DATA_BLOCK "DB_Output"	// DB 1010
AUTHOR : Broecker
VERSION : 0.1
  STRUCT
   Spare_A100_0 : BOOL ;
   Fuse_24V_DC_Reset : BOOL ;
   Spare_A100_2 : BOOL ;
   Spare_A100_3 : BOOL ;
   Spare_A100_4 : BOOL ;
   Status_LED_Bit0 : BOOL ;
   Status_LED_Bit1 : BOOL ;
   Status_LED_Bit2 : BOOL ;
   LED_Automatic : BOOL ;
   LED_Reset : BOOL ;
   Spare_A101_2 : BOOL ;
   Spare_A101_3 : BOOL ;
   Spare_A101_4 : BOOL ;
   Spare_A101_5 : BOOL ;
   Spare_A101_6 : BOOL ;
   Spare_A101_7 : BOOL ;
   Emergency_Stop_Reset : BOOL ;
   Spare_A102_1 : BOOL ;
   Spare_A102_2 : BOOL ;
   Spare_A102_3 : BOOL ;
   Spare_A102_4 : BOOL ;
   Spare_A102_5 : BOOL ;
   Spare_A102_6 : BOOL ;
   Spare_A102_7 : BOOL ;
   Spare_A103_0 : BOOL ;
   Spare_A103_1 : BOOL ;
   Spare_A103_2 : BOOL ;
   Spare_A103_3 : BOOL ;
   Spare_A103_4 : BOOL ;
   Spare_A103_5 : BOOL ;
   Spare_A103_6 : BOOL ;
   Spare_A103_7 : BOOL ;
   Spare_A104_0 : BOOL ;
   Spare_A104_1 : BOOL ;
   Spare_A104_2 : BOOL ;
   Spare_A104_3 : BOOL ;
   Spare_A104_4 : BOOL ;
   Spare_A104_5 : BOOL ;
   Spare_A104_6 : BOOL ;
   Spare_A104_7 : BOOL ;
   Spare_A105_0 : BOOL ;
   Spare_A105_1 : BOOL ;
   Spare_A105_2 : BOOL ;
   Spare_A105_3 : BOOL ;
   Spare_A105_4 : BOOL ;
   Spare_A105_5 : BOOL ;
   Spare_A105_6 : BOOL ;
   Spare_A105_7 : BOOL ;
   Spare_A106_0 : BOOL ;
   Spare_A106_1 : BOOL ;
   Spare_A106_2 : BOOL ;
   Spare_A106_3 : BOOL ;
   Spare_A106_4 : BOOL ;
   Spare_A106_5 : BOOL ;
   Spare_A106_6 : BOOL ;
   Spare_A106_7 : BOOL ;
   Spare_A107_0 : BOOL ;
   Spare_A107_1 : BOOL ;
   Spare_A107_2 : BOOL ;
   Spare_A107_3 : BOOL ;
   Spare_A107_4 : BOOL ;
   Spare_A107_5 : BOOL ;
   Spare_A107_6 : BOOL ;
   Spare_A107_7 : BOOL ;
   Spare_A108_0 : BOOL ;
   Spare_A108_1 : BOOL ;
   Spare_A108_2 : BOOL ;
   Spare_A108_3 : BOOL ;
   Spare_A108_4 : BOOL ;
   Spare_A108_5 : BOOL ;
   Spare_A108_6 : BOOL ;
   Spare_A108_7 : BOOL ;
   Spare_A109_0 : BOOL ;
   Spare_A109_1 : BOOL ;
   Spare_A109_2 : BOOL ;
   Spare_A109_3 : BOOL ;
   Spare_A109_4 : BOOL ;
   Spare_A109_5 : BOOL ;
   Spare_A109_6 : BOOL ;
   Spare_A109_7 : BOOL ;
   Spare_A110_0 : BOOL ;
   Fuse_24V_DC_Reset_VEH : BOOL ;
   Spare_A110_2 : BOOL ;
   LED_Reset_VEH : BOOL ;
   Sound_Generator : BOOL ;
   Status_LED_Bit0_VEH : BOOL ;
   Status_LED_Bit1_VEH : BOOL ;
   Status_LED_Bit2_VEH : BOOL ;
   Emergency_Stop_Reset_VEH : BOOL ;
   Spare_A111_1 : BOOL ;
   Spare_A111_2 : BOOL ;
   Spare_A111_3 : BOOL ;
   Scanner_On : BOOL ;
   Scanner_Field_A : BOOL ;
   Scanner_Field_B : BOOL ;
   Spare_A111_7 : BOOL ;
   Spare_A112_0 : BOOL ;
   Spare_A112_1 : BOOL ;
   Safety_Bar_Op : BOOL ;
   Safety_Bar_Cl : BOOL ;
   Spare_A112_4 : BOOL ;
   Spare_A112_5 : BOOL ;
   Spare_A112_6 : BOOL ;
   Spare_A112_7 : BOOL ;
  END_STRUCT ;	
BEGIN
END_DATA_BLOCK

ORGANIZATION_BLOCK OB 1
TITLE = "Main Program Sweep (Cycle)"
VERSION : 0.1
VAR_TEMP
  OB1_EV_CLASS : BYTE ;	//Bits 0-3 = 1 (Coming event), Bits 4-7 = 1 (Event class 1)
  OB1_SCAN_1 : BYTE ;	//1 (Cold restart scan 1 of OB 1), 3 (Scan 2-n of OB 1)
  OB1_PRIORITY : BYTE ;	//Priority of OB Execution
  OB1_OB_NUMBR : BYTE ;	//1 (Organization block 1, OB1)
  OB1_RESERVED_1 : BYTE ;	//Reserved for system
  OB1_RESERVED_2 : BYTE ;	//Reserved for system
  OB1_PREV_CYCLE : INT ;	//Cycle time of previous OB1 scan (milliseconds)
  OB1_MIN_CYCLE : INT ;	//Minimum cycle time of OB1 (milliseconds)
  OB1_MAX_CYCLE : INT ;	//Maximum cycle time of OB1 (milliseconds)
  OB1_DATE_TIME : DATE_AND_TIME ;	//Date and time OB1 started
END_VAR
BEGIN
// (block stored without names or comments; labels and parameter names are numbered)
END_ORGANIZATION_BLOCK

SYMBOL_TABLE
"IDB_Safe_Main"	DB 1	FB 1
"DB_TRO"	DB 2	DB 2
"DB_LIF"	DB 3	DB 3
"DB_TEL"	DB 4	DB 4
"DB_BRI"	DB 5	DB 5
"DB_ComGateway"	DB 10	DB 10
"IDB_FB2_TRO"	DB 12	FB 2
"IDB_FB2_LIF"	DB 13	FB 2
"IDB_FB21_TEL"	DB 14	FB 21
"DB_OrderBuffer"	DB 15	DB 15
"DB_IntentData"	DB 17	DB 17
"DB_TargetData"	DB 19	DB 19
"IDB_FB22"	DB 22	FB 22
"IDB_FB29"	DB 29	FB 29
"IDB_MasterInterface"	DB 33	FB 13
"DB_ANALOG"	DB 50	DB 50
"INOUT"	DB 80	DB 80
"DB_ActualHookdata"	DB 92	DB 92	// Hookdata of actual trollayposition
"Moves"	DB 101	DB 101
"InstanzDB PNIODiag"	DB 126	FB 126
"InstanzDB STATDiag"	DB 127	DB 127
"DB_Crane"	DB 130	DB 130
"DB_Steps"	DB 132	DB 132
"DB_CylinderTypes"	DB 133	DB 133
"IDB_FB190"	DB 190	FB 190
"IDB_FB190_2"	DB 191	FB 190
"IDB1_FB192"	DB 192	FB 192
"IDB1_FB192_2"	DB 193	FB 192
"TRO_Positions"	DB 200	DB 200
"BR01_TR01"	DB 201	DB 201
"BR01_TR02"	DB 202	DB 202
"BR01_TR03"	DB 203	DB 203
"BR01_TR04"	DB 204	DB 204
"BR01_TR05"	DB 205	DB 205
"BR01_TR06"	DB 206	DB 206
"BR01_TR07"	DB 207	DB 207
"BR01_TR08"	DB 208	DB 208
"BR01_TR09"	DB 209	DB 209
"BR01_TR10"	DB 210	DB 210
"BR01_TR11"	DB 211	DB 211
"BR02_TR01"	DB 212	DB 212
"BR02_TR02"	DB 213	DB 213
"BR02_TR03"	DB 214	DB 214
"BR02_TR04"	DB 215	DB 215
"BR02_TR05"	DB 216	DB 216
"BR02_TR06"	DB 217	DB 217
"BR02_TR07"	DB 218	DB 218
"BR02_TR08"	DB 219	DB 219
"BR02_TR09"	DB 220	DB 220
"BR02_TR10"	DB 221	DB 221
"BR02_TR11"	DB 222	DB 222
"BR03_TR01"	DB 223	DB 223
"BR03_TR02"	DB 224	DB 224
"BR03_TR03"	DB 225	DB 225
"BR03_TR04"	DB 226	DB 226
"BR03_TR05"	DB 227	DB 227
"BR03_TR06"	DB 228	DB 228
"BR03_TR07"	DB 229	DB 229
"BR03_TR08"	DB 230	DB 230
"BR03_TR09"	DB 231	DB 231
"BR03_TR10"	DB 232	DB 232
"BR03_TR11"	DB 233	DB 233
"BR04_TR01"	DB 234	DB 234
"BR04_TR02"	DB 235	DB 235
"BR04_TR03"	DB 236	DB 236
"BR04_TR04"	DB 237	DB 237
"BR04_TR05"	DB 238	DB 238
"BR04_TR06"	DB 239	DB 239
"BR04_TR07"	DB 240	DB 240
"BR04_TR08"	DB 241	DB 241
"BR04_TR09"	DB 242	DB 242
"BR04_TR10"	DB 243	DB 243
"BR04_TR11"	DB 244	DB 244
"BR05_TR01"	DB 245	DB 245
"BR05_TR02"	DB 246	DB 246
"BR05_TR03"	DB 247	DB 247
"BR05_TR04"	DB 248	DB 248
"BR05_TR05"	DB 249	DB 249
"BR05_TR06"	DB 250	DB 250
"BR05_TR07"	DB 251	DB 251
"BR05_TR08"	DB 252	DB 252
"BR05_TR09"	DB 253	DB 253
"BR05_TR10"	DB 254	DB 254
"BR05_TR11"	DB 255	DB 255
"BR06_TR01"	DB 256	DB 256
"BR06_TR02"	DB 257	DB 257
"BR06_TR03"	DB 258	DB 258
"BR06_TR04"	DB 259	DB 259
"BR06_TR05"	DB 260	DB 260
"BR06_TR06"	DB 261	DB 261
"BR06_TR07"	DB 262	DB 262
"BR06_TR08"	DB 263	DB 263
"BR06_TR09"	DB 264	DB 264
"BR06_TR10"	DB 265	DB 265
"BR06_TR11"	DB 266	DB 266
"BR07_TR01"	DB 267	DB 267
"BR07_TR02"	DB 268	DB 268
"BR07_TR03"	DB 269	DB 269
"BR07_TR04"	DB 270	DB 270
"BR07_TR05"	DB 271	DB 271
"BR07_TR06"	DB 272	DB 272
"BR07_TR07"	DB 273	DB 273
"BR07_TR08"	DB 274	DB 274
"BR07_TR09"	DB 275	DB 275
"BR07_TR10"	DB 276	DB 276
"BR07_TR11"	DB 277	DB 277
"BR08_TR01"	DB 278	DB 278
"BR08_TR02"	DB 279	DB 279
"BR08_TR03"	DB 280	DB 280
"BR08_TR04"	DB 281	DB 281
"BR08_TR05"	DB 282	DB 282
"BR08_TR06"	DB 283	DB 283
"BR08_TR07"	DB 284	DB 284
"BR08_TR08"	DB 285	DB 285
"BR08_TR09"	DB 286	DB 286
"BR08_TR10"	DB 287	DB 287
"BR08_TR11"	DB 288	DB 288
"BR09_TR01"	DB 289	DB 289
"BR09_TR02"	DB 290	DB 290
"BR09_TR03"	DB 291	DB 291
"BR09_TR04"	DB 292	DB 292
"BR09_TR05"	DB 293	DB 293
"BR09_TR06"	DB 294	DB 294
"BR09_TR07"	DB 295	DB 295
"BR09_TR08"	DB 296	DB 296
"BR09_TR09"	DB 297	DB 297
"BR09_TR10"	DB 298	DB 298
"BR09_TR11"	DB 299	DB 299
"BR10_TR01"	DB 300	DB 300
"BR10_TR02"	DB 301	DB 301
"BR10_TR03"	DB 302	DB 302
"BR10_TR04"	DB 303	DB 303
"BR10_TR05"	DB 304	DB 304
"BR10_TR06"	DB 305	DB 305
"BR10_TR07"	DB 306	DB 306
"BR10_TR08"	DB 307	DB 307
"BR10_TR09"	DB 308	DB 308
"BR10_TR10"	DB 309	DB 309
"BR10_TR11"	DB 310	DB 310
"BR11_TR01"	DB 311	DB 311
"BR11_TR02"	DB 312	DB 312
"LIF_Pos"	DB 350	DB 350
"IDB_Modbus1"	DB 362	FB 102
"ProfiNet"	DB 400	DB 400
"Error_Safety"	DB 410	DB 410
"IDB_ESTOP_1"	DB 450	FB 215
"IDB_ESTOP_2"	DB 451	FB 185
"IDB_Auto"	DB 452	FB 186
"F_GLOBDB"	DB 545	DB 545	// F_: F_Global_Data Block
"F00035_75x_667_4FDI_4FDO"	DB 555	FB 272
"F00040_75x_667_4FDI_4FDO"	DB 556	FB 272
"F00045_75x_661_4FDI_24V"	DB 557	FB 272
"F00055_75x_667_4FDI_4FDO"	DB 558	FB 272
"F_IO"	DB 690	DB 690
"F_Position"	DB 695	DB 695
"F_GBL_RECV"	DB 750	DB 750
"IDB_F_RCV"	DB 751	FB 226
"F_GBL_SEND"	DB 752	DB 752
"IDB_F_SND"	DB 753	FB 225
"IDB_WagoiPar_Rack"	DB 901	FB 37
"IDB_WagoiPar_BRI"	DB 920	FB 37
"IDB_WagoiPar_TRO"	DB 921	FB 37
"IDB_WagoiPar_LIF"	DB 922	FB 37
"DB_iPar_Diag"	DB 930	FB 101
"DIAG_PROFI_V2_iPar"	DB 931	DB 931	// diagnosis data of PROFIsafe modules V2 iPar with FB101
"DB_Vorlage"	DB 999	DB 999
"DB_LS1"	DB 1300	DB 1300
"IDB_LS1_Circum"	DB 1329	FB 29
"DB_LS"	DB 1350	DB 1350
"iPar_Data_Rack"	DB 1901	DB 1901
"iPar_Data_Bridge"	DB 1920	DB 1920
"iPar_Data_Trolley"	DB 1921	DB 1921
"iPar_Data_Lift"	DB 1922	DB 1922
"Safe_Main"	FB 1	FB 1
"MovidriveB_Control"	FB 2	FB 2
"MasterInterface"	FB 13	FB 13
"CheckEncoder"	FB 21	FB 21
"GetCircumference"	FB 22	FB 22
"WAGO_Analog_Input_4_20"	FB 29	FB 29	// WAGO A/D-Wandler 4-20mA
"WAGO_iPar_UDL_4_Mod"	FB 37	FB 37	// WAGO up- / download iParameter PROFIsafe Modules
"TSEND"	FB 63	FB 63	// Send Data
"TRCV"	FB 64	FB 64	// Receive Data
"TCON"	FB 65	FB 65	// Connect
"TDISCON"	FB 66	FB 66	// Disconnect
"Safety_Position"	FB 70	FB 70	// Sichere Positionsüberwachung
"Safety_Direction"	FB 72	FB 72	// Sichere Richtungserfassung
"Safety_Speed"	FB 73	FB 73	// Sichere Geschwindigkeit
"Safety_SpeedCheck"	FB 74	FB 74
"Wago_Trolley"	FB 81	FB 81
"F_Input_MAP"	FB 91	FB 91
"ESTOP"	FB 92	FB 92
"GetArea"	FB 95	FB 95
"DiagPROFIsafe_V2_iPar"	FB 101	FB 101	// read diagnosis data of PROFIsafe modules V2 iPar
"MODBUSPN"	FB 102	FB 102	// MODBUS PN CPU
"TCP_COMM"	FB 103	FB 103	// TCP Kommunikation
"MOD_CLI"	FB 104	FB 104
"MOD_SERV"	FB 105	FB 105
"PNIODiag"	FB 126	FB 126	// Profibus/DP und Profinet/IO-Diagnose
"STATDiag"	FB 127	FB 127	// Zweitbaustein (PNIODiag)
"F_TON"	FB 185	FB 185	// F_: Timer Switch On Delay
"F_TOF"	FB 186	FB 186	// F_: Timer Switch Off Delay
"CopyHookDBs"	FB 190	FB 190
"READ_DBL"	FB 192	FB 192	// read db from memorycard
"WRITE_DBL"	FB 193	FB 193	// write db to memorycard
"F_ESTOP1"	FB 215	FB 215	// F_: Emergency Stop / Stop Category 1
"F_ACK_GL"	FB 219	FB 219	// F_: Global Acknowledgement of all F-I/O of a RTG
"F_SENDS7"	FB 225	FB 225	// F_: Send S7 Connection
"F_RCVS7"	FB 226	FB 226	// F_: Receive S7 Connection
"F_IO_CGP"	FB 272	FB 272	// F_: Driver Block In-Output with Channel Granular Passivation
"F_CTRL_1"	FB 273	FB 273
"F_CTRL_2"	FB 274	FB 274	// F_: Test Block an Programm Run Control
"F_DIAG_N"	FB 275	FB 275
"FITON"	FB 276	FB 276
"FITOF"	FB 277	FB 277
"FIACK_GL"	FB 278	FB 278
"F-CALL"	FC 1	FC 1
"Init"	FC 2	FC 2
"AG_SEND"	FC 5	FC 5	// AG SEND
"AG_RECV"	FC 6	FC 6	// AG RECEIVE
"DT_TOD"	FC 8	FC 8	// DT to TOD
"OpHours"	FC 9	FC 9
"EQ_STRNG"	FC 10	FC 10	// Equal String
"AbsEncoder"	FC 11	FC 11
"Motor_2_frequ"	FC 12	FC 12
"DT to DATE"	FC 15	FC 15	// DT to DATE
"Scan_BRI"	FC 21	FC 21
"Scan_BRI_MAN"	FC 22	FC 22	// Scan Bride Manual Mode
"Scan_BRI_DBs"	FC 23	FC 23
"Scan_LIF"	FC 25	FC 25
"Scan_LIF_Man"	FC 26	FC 26
"Scan_TEL"	FC 27	FC 27
"Scan_TEL_Man"	FC 28	FC 28
"SCALE_WAGO_AI"	FC 29	FC 29	// for WAGO 250-466 4-20mA SE Standard
"Inputs"	FC 30	FC 30
"Outputs"	FC 31	FC 31
"MeasureSystem"	FC 33	FC 33
"SEL"	FC 36	FC 36	// Select
"Errors"	FC 40	FC 40
"Errors Reset"	FC 41	FC 41
"Errors_001-016_GEN1"	FC 42	FC 42
"Errors_017-032_GEN2"	FC 43	FC 43
"Errors_033-048_NET"	FC 44	FC 44
"Errors_113-128"	FC 45	FC 45
"Errors_129-144_08"	FC 46	FC 46
"Errors_145-160"	FC 47	FC 47
"EOff_MachineOff"	FC 48	FC 48
"OP_Mode"	FC 49	FC 49
"Send_Buffer"	FC 52	FC 52
"MSG_161-176"	FC 55	FC 55
"MSG_177_192"	FC 56	FC 56
"CableDrum"	FC 60	FC 60
"TargetPosLift"	FC 70	FC 70
"CheckHookType"	FC 72	FC 72
"CheckWindowDi"	FC 100	FC 100
"Communication"	FC 103	FC 103
"STEPS_Control"	FC 110	FC 110
"STEPS_OrderData"	FC 111	FC 111
"STEPS_BASEPOS"	FC 112	FC 112
"STEPS_EMPTY"	FC 113	FC 113
"STEPS_GET"	FC 114	FC 114
"STEPS_PUT"	FC 115	FC 115
"Axis_TROLLEY"	FC 210	FC 210
"Axis_TROLLEY_Release"	FC 211	FC 211
"Axis_TROLLEY_Control"	FC 212	FC 212
"Axis_TROLLEY_Speed"	FC 213	FC 213
"Axis_TROLLEY_Scan"	FC 214	FC 214
"Axis_TROLLEY_Scan_Man"	FC 215	FC 215
"Axis_TROLLEY_Flt_065-080"	FC 219	FC 219
"Axis_LIFT"	FC 220	FC 220
"Axis_LIFT_Control"	FC 222	FC 222
"Axis_LIFT_Speed"	FC 223	FC 223
"Axis_LIFT_Scan"	FC 224	FC 224
"Axis_LIFT_Flt_081-096"	FC 229	FC 229
"Axis_TELESCOPES"	FC 230	FC 230
"Axis_TEL_Control"	FC 232	FC 232
"Axis_TEL_Speed"	FC 233	FC 233
"Axis_TEL_Scan"	FC 234	FC 234
"Axis_TEL_Chk"	FC 235	FC 235
"Axis_TEL_Status"	FC 236	FC 236
"Axis_TEL_Mode_Status"	FC 237	FC 237
"Axis_TEL_BCD"	FC 238	FC 238
"Axis_TEL_Flt_097-112"	FC 239	FC 239
"Axis_TEL_Encoder"	FC 240	FC 240
"iPar_ServerCall"	FC 900	FC 900
"Scan_LIF_New"	FC 1025	FC 1025
"Scan_LIF_Man_New"	FC 1026	FC 1026
"TROGetPosVal"	FC 1071	FC 1071
"E   35.0"	I 35.0	BOOL	// spare
"E   35.1"	I 35.1	BOOL	// spare
"I_TRO_FB_Lift"	I 35.2	BOOL	// Feedback safestop lift
"I_TRO_FB_Trolley"	I 35.3	BOOL	// Feedback safestop  trolley
"I_TRO_FB_Telescope"	I 40.0	BOOL	// Feedback safestop no FU
"E   40.1"	I 40.1	BOOL	// spare
"I_TRO_FB_Estop_CH1"	I 40.2	BOOL	// Feedback E-Stop  CH1
"I_TRO_FB_Estop_CH2"	I 40.3	BOOL	// Feedback E-Stop  CH2
"I_TRO_EStop"	I 45.0	BOOL	// Emergency stop activ
"I_TRO_Brake_OK"	I 45.1	BOOL	// Temperature brake resistors OK
"E   45.2"	I 45.2	BOOL	// spare
"E   45.3"	I 45.3	BOOL	// spare
"I_TRO_LIF_Overl_L_NC"	I 55.0	BOOL	// Overload-Monitoring left NC
"I_TRO_LIF_Overl_R_NC"	I 55.1	BOOL	// Overload-Monitoring right NC
"I_TRO_LIF_Slap_L_NC"	I 55.2	BOOL	// Slap-Rope-Monitoring left NC
"I_TRO_LIF_Slap_R_NC"	I 55.3	BOOL	// Slap-Rope-Monitoring right NC
"I_TRO_Fuse_115V_OK"	I 75.0	BOOL	// 115V AC OK
"I_TRO_Fuse_24V_OK"	I 75.1	BOOL	// fuse 24V DC OK
"I_TRO_Overtemp_Cabinet"	I 75.2	BOOL	// high temperature cabinet
"I_TRO_Power Brakes_OK"	I 75.3	BOOL	// Power supply brakes OK
"I_TRO_Power_Lift_OK"	I 75.4	BOOL	// Power supply lift OK
"I_TRO_Power_Drum_OK"	I 75.5	BOOL	// Power supply cable drum OK
"I_TRO_Power_Cabinet_Fan"	I 75.6	BOOL	// Power supply cabinet fan OK
"I_TRO_Cabinet_Fan_On"	I 75.7	BOOL	// cabinet fan running
"I_TRO_BTN_Reset"	I 76.0	BOOL	// Reset button (top cabinet)
"I_TRO_BTN_Preset"	I 76.1	BOOL	// Preset button (3s)
"I_TRO_Preset_Bit_0"	I 76.2	BOOL	// Preset selection switch bit 0
"I_TRO_Preset_Bit_1"	I 76.3	BOOL	// Preset selection switch bit 1
"I_TRO_Preset_Bit_2"	I 76.4	BOOL	// Preset selection switch bit 2
"I_TRO_Preset_Bit_3"	I 76.5	BOOL	// Preset selection switch bit 3
"E 76_6"	I 76.6	BOOL	// spare
"E 76_7"	I 76.7	BOOL	// spare
"I_Check_CableDrum_NO"	I 77.0	BOOL	// check cable drum NO
"I_Check_CableDrum_NC"	I 77.1	BOOL	// check cable drum NC
"E  77_2"	I 77.2	BOOL	// spar
"E  77_3"	I 77.3	BOOL	// spar
"I_Buffer_left_Free"	I 77.4	BOOL	// Buffer left occupied //
"I_Buffer_right_Free"	I 77.5	BOOL	// Buffer right occupied //
"I_LIF_Limit_TOP"	I 77.6	BOOL	// Lift limit switch top (minus)
"I_LIF_Limit_BOTTOM"	I 77.7	BOOL	// Lift limit switch bottom (plus)
"I_LIF_Pos_TOP_NO"	I 78.0	BOOL	// Lift limit prox. top NO
"I_LIF_Pos_TOP_NC"	I 78.1	BOOL	// Lift limit prox. top NC
"I_TRO_Limit_plus"	I 78.2	BOOL	// Tolley limit switch plus
"I_TRO_Limit_minus"	I 78.3	BOOL	// Tolley limit switch minus
"I_TRO_FS_plus_NO"	I 78.4	BOOL	// Tolley prox. switch forced slow plus NO
"I_TRO_FS_plus_NC"	I 78.5	BOOL	// Tolley prox. switch forced slow plus NC
"I_TRO_FS_minus_NO"	I 78.6	BOOL	// Tolley prox. switch forced slow minus NO
"I_TRO_FS_minus_NC"	I 78.7	BOOL	// Tolley prox. switch forced slow minus NC
"I_SSI_Barcode_noPos"	I 79.0	BOOL	// Datamatrix SSI error: no position
"I_SSI_Barcode_dirty"	I 79.1	BOOL	// Datamatrix SSI error: dirty
"I_Profinet_Barcode_noPos"	I 79.2	BOOL	// Datamatrix Profinet error: no position
"I_Profinet_Barcode_dirty"	I 79.3	BOOL	// Datamatrix Profinet error: dirty
"I_TRO_Drop_1_P"	I 79.4	BOOL	// Trolley drop off protection plus 1
"I_TRO_Drop_2_P"	I 79.5	BOOL	// Trolley drop off protection plus 2
"I_TRO_Drop_1_M"	I 79.6	BOOL	// Trolley drop off protection minus 1
"I_TRO_Drop_2_M"	I 79.7	BOOL	// Trolley drop off protection minus 2
"I_TRO_Plus"	I 80.0	BOOL	// Trolley drive plus
"I_TRO_Minus"	I 80.1	BOOL	// Trolley drive minus
"I_Lift_up"	I 80.2	BOOL	// Lift drive up
"I_Lift_down"	I 80.3	BOOL	// Lift drive down
"I_TEL_Plus"	I 80.4	BOOL	// Tellescope drive plus
"I_TEL_Minus"	I 80.5	BOOL	// Telescope drive minus
"E 80_6"	I 80.6	BOOL	// spare
"E 80_7"	I 80.7	BOOL	// spare
"E 85_0"	I 85.0	BOOL	// spare
"E 85_1"	I 85.1	BOOL	// spare
"E 85_2"	I 85.2	BOOL	// spare
"E 85_3"	I 85.3	BOOL	// spare
"I_TEL_Status1"	I 85.4	BOOL	// Drive telescopes status1
"I_TEL_Status2"	I 85.5	BOOL	// Drive telescopes status2
"E 85_6"	I 85.6	BOOL
"E 85_7"	I 85.7	BOOL
"I_LIF_Overload_L_NO"	I 86.0	BOOL	// Overload-Monitoring left NO
"I_LIF_Overload_R_NO"	I 86.1	BOOL	// Overload-Monitoring right NO
"I_LIF_SlapRope_L_NO"	I 86.2	BOOL	// Slap-Rope-Monitoring left NO
"I_LIF_SlapRope_R_NO"	I 86.3	BOOL	// Slap-Rope-Monitoring right NO
"E      86.4"	I 86.4	BOOL	// spare
"E      86.5"	I 86.5	BOOL	// spare
"I_LIF_Front_LastHookOcc"	I 86.6	BOOL	// hook front left occupied long
"I_LIF_Front_FirstHookOcc"	I 86.7	BOOL	// hook rear left occupied short
"I_LIF_Rear_LastHookOcc"	I 87.0	BOOL	// hook front right occupied long
"I_LIF_Rear_FirstHookOcc"	I 87.1	BOOL	// hook rear right occupied short
"E      87.2"	I 87.2	BOOL	// spare
"E      87.3"	I 87.3	BOOL	// spare
"I_TEL_inMidle_L"	I 87.4	BOOL	// telescope left in middle position
"I_TEL_inMidle_R"	I 87.5	BOOL	// telescope right in middle position
"E      87.6"	I 87.6	BOOL
"I_TEL_Left_Occ_NO"	I 87.7	BOOL	// telescope left occupied NO
"E      88.0"	I 88.0	BOOL
"I_TEL_Right_Occ_NO"	I 88.1	BOOL	// telescope right occupied NO
"I_TEL_Limit_front_NO"	I 88.2	BOOL	// telescopes limit switch front NO
"I_TEL_Limit_front_NC"	I 88.3	BOOL	// telescopes limit switch front NC
"I_TEL_Limit_back_NO"	I 88.4	BOOL	// telescopes limit switch back NO
"I_TEL_Limit_back_NC"	I 88.5	BOOL	// telescopes limit switch back NC
"E      88.6"	I 88.6	BOOL	// spare
"E      88.7"	I 88.7	BOOL	// spare
"E      89.0"	I 89.0	BOOL
"E      89.1"	I 89.1	BOOL
"E      89.2"	I 89.2	BOOL
"E      89.3"	I 89.3	BOOL
"E      89.4"	I 89.4	BOOL
"E      89.5"	I 89.5	BOOL
"E      89.6"	I 89.6	BOOL
"E      89.7"	I 89.7	BOOL
"OFF"	M 0.0	BOOL	// immer aus
"ON"	M 0.1	BOOL	// immer ein
"TRUE"	M 0.2	BOOL
"FALSE"	M 0.3	BOOL
"FIRST_RUN"	M 0.7	BOOL
"ModeService"	M 1.0	BOOL
"ModeManual"	M 1.1	BOOL
"ModeAuto"	M 1.2	BOOL
"ModeBypass"	M 1.3	BOOL
"ModeServiceOrManual"	M 1.4	BOOL
"SEW_EmergencyMode"	M 1.5	BOOL
"ModeAutoOrManual"	M 1.6	BOOL
"LifeBitMasterOK"	M 1.7	BOOL
"Eoff"	M 2.0	BOOL
"DivEoff"	M 2.1	BOOL
"Error"	M 2.2	BOOL
"EmOffRelais_delayed"	M 3.0	BOOL
"TRO_pFL_StopOnCarrier"	M 8.0	BOOL
"TRO_StopOnCarrier"	M 8.1	BOOL
"LIF_pFl_manPrevPos"	M 9.0	BOOL
"LIF_pFl_manNextPos"	M 9.1	BOOL
"Tel_pFl_manMinusPos"	M 9.2	BOOL
"Tel_pFl_manPlusPos"	M 9.3	BOOL
"TEL_nFl_CenterPos"	M 9.4	BOOL
"TEL_StopInCenter"	M 9.5	BOOL
"TEL_pFl_StopInCenter"	M 9.6	BOOL
"Clock0_1"	M 10.0	BOOL	// CPU-Takt 0,1s
"Clock0_2"	M 10.1	BOOL	// CPU-Takt 0,2s
"Clock0_4"	M 10.2	BOOL	// CPU-Takt 0,4s
"Clock0_5"	M 10.3	BOOL	// CPU-Takt 0,5s
"Clock0_8"	M 10.4	BOOL	// CPU-Takt 0,8s
"Clock1_0"	M 10.5	BOOL	// CPU-Takt 1,0s
"Clock1_6"	M 10.6	BOOL	// CPU-Takt 1,6s
"Clock2_0"	M 10.7	BOOL	// CPU-Takt 2,0s
"Tick0_1"	M 11.0	BOOL	// Impuls 0,1s
"Tick0_2"	M 11.1	BOOL	// Impuls 0,2s
"Tick0_4"	M 11.2	BOOL	// Impuls 0,4s
"Tick0_5"	M 11.3	BOOL	// Impuls 0,6s
"Tick0_8"	M 11.4	BOOL	// Impuls 0,8s
"Tick1_0"	M 11.5	BOOL	// Impuls 1,0s
"Tick1_6"	M 11.6	BOOL	// Impuls 1,6s
"Tick2_0"	M 11.7	BOOL	// Impuls 2,0s
"SysPulse_0_1"	M 12.0	BOOL
"SysPulse_0_2"	M 12.1	BOOL
"SysPulse_0_4"	M 12.2	BOOL
"SysPulse_0_5"	M 12.3	BOOL
"SysPulse_0_8"	M 12.4	BOOL
"SysPulse_1_0"	M 12.5	BOOL
"SysPulse_1_6"	M 12.6	BOOL
"SysPulse_2_0"	M 12.7	BOOL
"StartModeAuto"	M 13.0	BOOL
"TEL_pFl_Start"	M 19.0	BOOL
"NullBit"	M 20.0	BOOL
"CB_Lamp_Preset"	M 21.0	BOOL
"TEL_Save_Long_POS_front"	M 25.0	BOOL
"TEL_Save_Long_POS_rear"	M 25.1	BOOL
"TrolleyWasOnCarrier"	M 40.0	BOOL
"SendTrolleyWasOnCarrier"	M 40.1	BOOL
"Next_Step"	M 44.0	BOOL
"SingleStep_ON"	M 44.1	BOOL
"One_Single_Step"	M 44.2	BOOL
"TEL_RackPos"	M 55.0	BOOL
"TEL_LS1_Pos"	M 55.1	BOOL
"TEL_LS2_Pos"	M 55.2	BOOL
"TEL_LS3_Pos"	M 55.3	BOOL
"Safety_Tele_Center"	M 152.0	BOOL
"Safety_Tele_Rear"	M 152.1	BOOL
"Safety_Tele_Front"	M 152.2	BOOL
"Safety_Trolley_in_Pos"	M 153.0	BOOL
"Safety_Lift_Top"	M 154.0	BOOL
"Safety_Lift_Over"	M 154.1	BOOL
"Safety_Lift_Under"	M 154.2	BOOL
"Mode_Bypass"	M 200.2	BOOL
"RED_IBN_Test"	M 420.0	BOOL
"IBN_1"	M 500.0	BOOL
"IBN_0"	M 500.1	BOOL
"TRO_iPar_Check"	M 921.0	BOOL
"TRO_iPar_UpLoad"	M 921.1	BOOL
"TRO_iPar_DownL"	M 921.2	BOOL
"TRO_iPar_ReqDiag"	M 921.5	BOOL
"LIF_iPar_Check"	M 922.0	BOOL
"LIF_iPar_UpLoad"	M 922.1	BOOL
"LIF_iPar_DownL"	M 922.2	BOOL
"LIF_iPar_ReqDiag"	M 922.5	BOOL
"TRO_pFl_iPar"	M 925.1	BOOL
"LIF_pFl_iPar_1"	M 925.2	BOOL
"LIF_pFl_iPar_2"	M 925.3	BOOL
"PowerFan_pl"	M 1001.0	BOOL
"PowerFan_n"	M 1001.1	BOOL
"P_FL_TeleCheck1"	M 1401.2	BOOL
"N_FL_TeleCheck1"	M 1401.3	BOOL
"P_FL_TeleCheck2"	M 1401.6	BOOL
"N_FL_TeleCheck2"	M 1401.7	BOOL
"TeleCheckErr1"	M 1402.0	BOOL
"TeleCheckErr2"	M 1402.1	BOOL
"TeleCheckErr3"	M 1402.3	BOOL
"TeleCheckErr4"	M 1402.4	BOOL
"Reset_Err"	M 1410.0	BOOL
"Impuls_1"	M 1500.0	BOOL
"Impuls_2"	M 1500.1	BOOL
"Impuls_3"	M 1500.2	BOOL
"Impuls_4"	M 1500.3	BOOL
"Impuls_5"	M 1500.4	BOOL
"Impuls_6"	M 1500.5	BOOL
"Impuls_7"	M 1500.6	BOOL
"Impuls_8"	M 1500.7	BOOL
"Bruno_B1"	M 2013.0	BOOL	// Programmpunkt muss noch bearbeitet werden
"Bruno_B2"	M 2013.1	BOOL	// Schmiermerker
"TEL_SaveTarget"	MW 14	INT
"NullWord"	MW 20	WORD
"PC_MSG_Counter"	MW 120	INT
"Bruno_W1"	MW 2014	WORD	// Schmierwort
"Bruno_W2"	MW 2016	WORD	// Schmierwort
"CYCL_EXC"	OB 1	OB 1
"CYC_INT5"	OB 35	OB 35	// Cyclic Interrupt 5
"CYCL_FLT"	OB 80	OB 80	// Cycle Time Fault
"I/O_FLT1"	OB 82	OB 82	// I/O Point Fault 1
"I/O_FLT2"	OB 83	OB 83	// I/O Point Fault 2
"OBNL_FLT"	OB 85	OB 85	// OB Not Loaded Fault
"RACK_FLT"	OB 86	OB 86	// Loss of Rack Fault
"COMM_FLT"	OB 87	OB 87	// Communication Fault
"STARTUP"	OB 100	OB 100
"PROG_ERR"	OB 121	OB 121	// Programming Error
"MOD_ERR"	OB 122	OB 122	// Module Access Error
"O_Bypass_RC"	Q 35.0	BOOL	// bypass remote control
"A    35.1"	Q 35.1	BOOL	// spare
"O_SafeStop_Lift"	Q 35.2	BOOL	// safe stop lift
"O_SafeStop_Trolley"	Q 35.3	BOOL	// safe stop trolley
"O_SafeStop_Telecope"	Q 40.0	BOOL	// safe stop telescope
"A    40.1"	Q 40.1	BOOL	// spare
"O_TRO_Stop_CH1"	Q 40.2	BOOL	// E-Stop trolley CH1
"O_TRO_Stop_CH2"	Q 40.3	BOOL	// E-Stop trolley CH2
"O_SafeRelease_Telescope"	Q 55.0	BOOL
"A 75_0"	Q 75.0	BOOL	// spare
"O_TRO_Reset_24V"	Q 75.1	BOOL	// reset 24V fuses
"A 75_2"	Q 75.2	BOOL	// spare
"O_TRO_LP_Reset"	Q 75.3	BOOL	// lamp reset
"A 75_4"	Q 75.4	BOOL	// spare
"O_TRO_CableDrum"	Q 75.5	BOOL	// start cable drum
"O_TRO_EStop_Reset"	Q 75.6	BOOL	// ESTOP reset
"O_TRO_LP_Preset"	Q 75.7	BOOL	// lamp preset
"O_TRO_Horn"	Q 76.0	BOOL	// startup warning
"O_TRO_State_0"	Q 76.1	BOOL	// lamp state 0
"O_TRO_State_1"	Q 76.2	BOOL	// lamp state 1
"O_TRO_state_2"	Q 76.3	BOOL	// lamp state 2
"A      76.4"	Q 76.4	BOOL	// spare
"O_TRO_MoviPLC_Reset"	Q 76.5	BOOL	// reset movi PLC
"O_TRO_EmergencyMode"	Q 76.6	BOOL	// Emergency Mode
"O_LIFT_StartFan"	Q 76.7	BOOL	// start Lift Fan
"O_TRO_EmergencyMode_Fwd"	Q 77.0	BOOL	// Emergency mode forward
"O_TRO_EmergencyMode_Bwd"	Q 77.1	BOOL	// Emergency mode backward
"A      77.2"	Q 77.2	BOOL
"A      77.3"	Q 77.3	BOOL
"A      77.4"	Q 77.4	BOOL
"A      77.5"	Q 77.5	BOOL
"A      77.6"	Q 77.6	BOOL
"A      77.7"	Q 77.7	BOOL
"O_TEL_Mode1"	Q 85.0	BOOL	// telescope mode_1 Service
"O_TEL_Mode2"	Q 85.1	BOOL	// telescope mode_2 Automatic
"O_TEL_Start"	Q 85.2	BOOL	// start telescope
"O_TEL_Reset"	Q 85.3	BOOL	// reset telescope
"O_TEL_BCD_Bit_1"	Q 85.4	BOOL	// telescope BCD Bit_1
"O_TEL_BCD_Bit_2"	Q 85.5	BOOL	// telescope BCD Bit_2
"O_TEL_BCD_Bit_3"	Q 85.6	BOOL	// telescope BCD Bit_3
"O_TEL_BCD_Bit_4"	Q 85.7	BOOL	// telescope BCD Bit_4
"O_TEL_LightFront_Left"	Q 86.0	BOOL	// lightning telescopes front left ON
"O_TEL_LightFront_Right"	Q 86.1	BOOL	// lightning telescopes rear rigth ON
"O_TEL_LightRear_Left"	Q 86.2	BOOL	// lightning telescopes rear left ON
"O_TEL_LightRear_Right"	Q 86.3	BOOL	// lightning telescopes rear rigth ON
"O_TEL_Preset_Encoder"	Q 86.4	BOOL	// Preset Encoder Telescope
"A     86.5"	Q 86.5	BOOL	// spare
"A     86.6"	Q 86.6	BOOL	// spare
"A     86.7"	Q 86.7	BOOL	// spare
"A     87.0"	Q 87.0	BOOL
"A     87.1"	Q 87.1	BOOL
"A     87.2"	Q 87.2	BOOL
"A     87.3"	Q 87.3	BOOL
"A     87.4"	Q 87.4	BOOL
"A     87.5"	Q 87.5	BOOL
"A     87.6"	Q 87.6	BOOL
"A     87.7"	Q 87.7	BOOL
"TON"	SFB 4	SFB 4	// Generate an On Delay
"USEND"	SFB 8	SFB 8	// Uncoordinated Sending of Data
"URCV"	SFB 9	SFB 9	// Uncoordinated Receiving of Data
"RDREC"	SFB 52	SFB 52	// Read a Process Data Record
"WRREC"	SFB 53	SFB 53	// Write a Process Data Record
"RALRM"	SFB 54	SFB 54	// Receive Alarm Data
"DPRD_DAT"	SFC 14	SFC 14	// Read Consistent Data of a Standard DP Slave
"DPWR_DAT"	SFC 15	SFC 15	// Write Consistent Data to a Standard DP Slave
"BLKMOV"	SFC 20	SFC 20	// Copy Variables
"FILL"	SFC 21	SFC 21	// Initialize a Memory Area
"TEST_DB"	SFC 24	SFC 24	// Test Data Block
"DIS_AIRT"	SFC 41	SFC 41	// Delay the Higher Priority Interrupts and Asynchronous Errors
"EN_AIRT"	SFC 42	SFC 42	// Enable Higher Priority Interrupts and Asynchronous Errors
"STP"	SFC 46	SFC 46	// Change the CPU to STOP
"RDSYSST"	SFC 51	SFC 51	// Read a System Status List or Partial List
"WR_REC"	SFC 58	SFC 58	// Write Data Record
"RD_REC"	SFC 59	SFC 59	// Read a Data Record
"RD_DBL"	SFC 83	SFC 83	// Read Data Block from Load Memory
"WRIT_DBL"	SFC 84	SFC 84	// Write Data Block in Load Memory
"tPlcOn"	T 1	TIMER
"tAknowl"	T 2	TIMER
"tTimeout_TRO"	T 26	TIMER
"T_TRO_Preset"	T 30	TIMER
"tTimeout_LIF"	T 36	TIMER
"tTimeout_LIF2"	T 37	TIMER
"T_Startup_Warning"	T 94	TIMER
"T_Delay_Emeg_Mode"	T 110	TIMER
"T_Err_TR_Forced_minus"	T 152	TIMER
"T_Err_TR_Forced_plus"	T 153	TIMER
"T_CheckUS"	T 160	TIMER
"T_CheckUS_OK"	T 161	TIMER
"UDT_Any"	UDT 1	UDT 1
"UDT_SysSave"	UDT 2	UDT 2
"OneMove"	UDT 7	UDT 7
"UDT_SEWState"	UDT 11	UDT 11
"UDT_SEWControl"	UDT 12	UDT 12
"TrDataSheet"	UDT 20	UDT 20	// Zuordnung Turm-DBs
"TRODataSheet"	UDT 21	UDT 21
"HookData"	UDT 100	UDT 100
"HookDataSheetNeu"	UDT 101	UDT 101
"HookDataSheet"	UDT 102	UDT 102
"UDT_CylinderType"	UDT 110	UDT 110
"ROW5"	VAT 1	
"IO-Check"	VAT 2	
"ROW4"	VAT 3	
"ROW3"	VAT 4	
"ROW2"	VAT 5	
"ROW1"	VAT 6	
"ROW6"	VAT 7	
"Order"	VAT 8	
"VAT_Sonar"	VAT 9	
"VAT_Bruno"	VAT 10	
"VAT_NewTarget"	VAT 11	
"VAT_TEL_Encoder"	VAT 12	
"VAT_TR_POS_TEST"	VAT 13	
END_SYMBOL_TABLE

SYMBOL_TABLE
"IDB_SafeMain"	DB 1	FB 1
"CONTROL_DAT_1"	DB 2	DB 2
"License_DB"	DB 3	DB 3
"IDB_SafePosition"	DB 5	FB 2
"DATA_AREA_1"	DB 11	DB 11
"DATA_AREA_2"	DB 12	DB 12
"DATA_AREA_3"	DB 13	DB 13
"DATA_AREA_4"	DB 14	DB 14
"DATA_AREA_5"	DB 15	DB 15
"DATA_AREA_6"	DB 16	DB 16
"Remote1"	DB 25	DB 25
"iDB_FB29"	DB 29	FB 29
"iDB_LS2_Masterinterface"	DB 33	FB 13
"iDB_LS1_Masterinterface"	DB 34	FB 13
"IDB_FB35_Doors"	DB 35	FB 35
"INOUT"	DB 80	DB 80
"Global_Signals"	DB 90	DB 90
"LS1_Moves"	DB 103	DB 103
"LS2_Moves"	DB 104	DB 104
"iDB_UDP_COM"	DB 120	FB 120
"InstanzDB PNIODiag"	DB 126	FB 126
"InstanzDB STATDiag"	DB 127	DB 127
"DB_Steps_LS1"	DB 130	DB 130
"DB_Steps_LS2"	DB 131	DB 131
"COMM_CAR01"	DB 150	DB 150
"COMM_CAR02"	DB 151	DB 151
"COMM_TR01"	DB 152	DB 152
"COMM_TR02"	DB 153	DB 153
"COMM_TR03"	DB 154	DB 154
"COMM_LS01"	DB 155	DB 155
"COMM_LS02"	DB 156	DB 156
"COMM_LS03"	DB 157	DB 157
"COMM_MAIN"	DB 159	DB 159
"IDB_PUT"	DB 160	FB 15
"IDB_GET"	DB 161	FB 14
"iDB_LS1_Table_Lift"	DB 172	FB 172
"iDB_LS1_Table_left_right"	DB 173	FB 173
"iDB_LS1_Shuttle"	DB 174	FB 174
"Mode"	DB 180	DB 180
"Pipe_Magazin"	DB 200	DB 200
"iDB_Robotcontrol"	DB 210	FB 210
"PLC_to_Robot"	DB 250	DB 250
"Robot_to_PLC"	DB 251	DB 251
"iDB_LS2_Table_Lift"	DB 275	FB 175
"iDB_LS2_Table_left_right"	DB 276	FB 176
"iDB_LS2_Shuttle"	DB 277	FB 177
"DB_Modbus_Parameter1"	DB 300	DB 300
"IDB_Modbus1"	DB 302	FB 102
"ProfiNet"	DB 400	DB 400
"F_GLOBDB"	DB 545	DB 545	// F_: F_Global_Data Block
"F_IO"	DB 690	DB 690
"SafetyError"	DB 710	DB 710
"F_GBL_RCV1"	DB 750	DB 750
"IDB_F_RCV1"	DB 751	FB 226
"F_GBL_RCV2"	DB 752	DB 752
"IDB_F_RCV2"	DB 753	FB 226
"F_GBL_RCV3"	DB 754	DB 754
"IDB_F_RCV3"	DB 755	FB 226
"F_GBL_RCV4"	DB 756	DB 756
"IDB_F_RCV4"	DB 757	FB 226
"F_GBL_RCV5"	DB 758	DB 758
"IDB_F_RCV5"	DB 759	FB 226
"F_GBL_SND1"	DB 760	DB 760
"IDB_F_SND1"	DB 761	FB 225
"F_GBL_SND2"	DB 762	DB 762
"IDB_F_SND2"	DB 763	FB 225
"F_GBL_SND3"	DB 764	DB 764
"IDB_F_SND3"	DB 765	FB 225
"F_GBL_SND4"	DB 766	DB 766
"IDB_F_SND4"	DB 767	FB 225
"F_GBL_SND5"	DB 768	DB 768
"IDB_F_SND5"	DB 769	FB 225
"IDB_WagoiPar_CB_1"	DB 920	FB 37
"IDB_WagoiPar_CB_2"	DB 921	FB 37
"DB_iPar_Diag"	DB 930	FB 101
"IDB_WagoiPar_IO_1"	DB 940	FB 37
"IDB_WagoiPar_IO_2"	DB 941	FB 37
"F00270_8FDI_iPar___UINT8"	DB 1099	FB 545
"F00265_8FDI_iPar___UINT8"	DB 1100	FB 545
"F00250_4FDI_4FDO_iPar__"	DB 1101	FB 545
"F00255_4FDI_4FDO_iPar__"	DB 1102	FB 545
"F00000_PS_8_bytes"	DB 1103	FB 545
"F00260_8FDI_iPar___UINT8"	DB 1104	FB 545
"F00240_8FDI_iPar___UINT8"	DB 1106	FB 545
"F00235_8FDI_iPar___UINT8"	DB 1107	FB 545
"F00230_8FDI_iPar___UINT8"	DB 1108	FB 545
"F00225_8FDI_iPar___UINT8"	DB 1109	FB 545
"F00220_4FDI_4FDO_iPar__"	DB 1110	FB 545
"F00275_8FDI_iPar___UINT8"	DB 1123	FB 545
"ValuesRack"	DB 1400	DB 1400
"iPar_Data_CB_1"	DB 1920	DB 1920
"iPar_Data_CB_2"	DB 1921	DB 1921
"iPar_Data_CB_IO_1"	DB 1940	DB 1940
"iPar_Data_CB_IO_2"	DB 1941	DB 1941
"SafeMain"	FB 1	FB 1
"SafePosition"	FB 2	FB 2
"FB_DoorSwitch_Euchner"	FB 10	FB 10
"MasterInterface"	FB 13	FB 13
"GET"	FB 14	FB 14	// Read Data From a Remote CPU
"PUT"	FB 15	FB 15	// Write Data to a Remote CPU
"WAGO_Analog_Input_4_20"	FB 29	FB 29	// WAGO A/D-Wandler 4-20mA
"FB_Doors"	FB 35	FB 35
"WAGO_iPar_UDL_4_Mod"	FB 37	FB 37	// WAGO up- / download iParameter PROFIsafe Modules
"TSEND"	FB 63	FB 63	// Send Data
"TRCV"	FB 64	FB 64	// Receive Data
"TCON"	FB 65	FB 65	// Connect
"TDISCON"	FB 66	FB 66	// Disconnect
"Wago_Main"	FB 82	FB 82
"Wago_LS12"	FB 83	FB 83
"F_Input_MAP"	FB 91	FB 91
"ESTOP"	FB 92	FB 92
"STATION_12"	FB 93	FB 93
"DiagPROFIsafe_V2_iPar"	FB 101	FB 101	// read diagnosis data of PROFIsafe modules V2 iPar
"MODBUSPN"	FB 102	FB 102	// MODBUS PN CPU
"TCP_COMM"	FB 103	FB 103	// TCP Kommunikation
"MOD_CLI"	FB 104	FB 104
"MOD_SERV"	FB 105	FB 105
"UDP_Comm"	FB 120	FB 120
"PNIODiag"	FB 126	FB 126	// Profibus/DP und Profinet/IO-Diagnose
"STATDiag"	FB 127	FB 127	// Zweitbaustein (PNIODiag)
"LS1_Table_Lift"	FB 172	FB 172
"LS1_Table_left_right"	FB 173	FB 173
"LS1_Shutlle"	FB 174	FB 174
"LS2_Table_Lift"	FB 175	FB 175
"LS2_Table_left_right"	FB 176	FB 176
"LS2_Shutlle"	FB 177	FB 177
"F_TON"	FB 185	FB 185	// F_: Timer Switch On Delay
"F_TOF"	FB 186	FB 186	// F_: Timer Switch Off Delay
"Robot_Control"	FB 210	FB 210
"F_ESTOP1"	FB 215	FB 215	// F_: Emergency Stop / Stop Category 1
"F_ACK_GL"	FB 219	FB 219	// F_: Global Acknowledgement of all F-I/O of a RTG
"F_SENDS7"	FB 225	FB 225	// F_: Send S7 Connection
"F_RCVS7"	FB 226	FB 226	// F_: Receive S7 Connection
"F_IO_CGP"	FB 545	FB 545
"F_CTRL_1"	FB 546	FB 546
"F_CTRL_2"	FB 547	FB 547
"F_DIAG_N"	FB 548	FB 548	// F_: Diagnosticbuffer Message with non CPU-Stop
"FITON"	FB 549	FB 549
"FITOF"	FB 550	FB 550
"FIACK_GL"	FB 551	FB 551
"ModeSelect"	FB 720	FB 720
"F-CALL"	FC 1	FC 1
"Init"	FC 2	FC 2
"AG_SEND"	FC 5	FC 5	// AG SEND
"AG_RECV"	FC 6	FC 6	// AG RECEIVE
"DT_TOD"	FC 8	FC 8	// DT to TOD
"EQ_STRNG"	FC 10	FC 10	// Equal String
"DT to DATE"	FC 15	FC 15	// DT to DATE
"RemoteControlCrtl"	FC 20	FC 20
"RemoteControlValues"	FC 21	FC 21
"RemoteConrolLamps"	FC 22	FC 22
"RemoteControlError"	FC 23	FC 23
"RemoteStatus"	FC 24	FC 24
"RemoteControlButtons"	FC 25	FC 25
"Comm_Modbus1"	FC 27	FC 27
"SCALE_WAGO_AI"	FC 29	FC 29	// for WAGO 250-466 4-20mA SE Standard
"Inputs"	FC 30	FC 30
"Outputs"	FC 31	FC 31
"LS1_Errors"	FC 40	FC 40
"LS1_Errors Reset"	FC 41	FC 41
"LS1_Errors_001-016_GEN1"	FC 42	FC 42
"LS1_Errors_017-032_GEN2"	FC 43	FC 43
"LS1_Errors_033-048_CAB"	FC 44	FC 44
"LS1_EOff_MachineOff"	FC 48	FC 48
"LS1_OP_Mode"	FC 49	FC 49
"Send_Buffer"	FC 52	FC 52
"CB_Errors"	FC 70	FC 70
"CB_Errors_1_16"	FC 80	FC 80
"CB_Errors_17_32"	FC 81	FC 81
"CB_Errors_33_48"	FC 82	FC 82
"CB_Errors_49_64"	FC 83	FC 83
"CB_Errors_65_80"	FC 84	FC 84
"CB_Errors_80_96"	FC 85	FC 85
"CB_Errors_97_112"	FC 86	FC 86
"CB_Messages_113_128"	FC 87	FC 87
"CB_Messages_129_144"	FC 88	FC 88
"CB_Messages_145_160"	FC 89	FC 89
"LS1_STEPS_PALLETT_CHANGE"	FC 92	FC 92
"LS1_Communication"	FC 103	FC 103
"LS2_Communication"	FC 104	FC 104
"LS1_Errors_081-096"	FC 130	FC 130
"LS1_OP_161_176"	FC 135	FC 135
"LS2_Errors"	FC 140	FC 140
"LS2_Errors Reset"	FC 141	FC 141
"LS2_Errors_001-016_GEN1"	FC 142	FC 142
"LS2_Errors_017-032_GEN2"	FC 143	FC 143
"LS2_Errors_033-048_CAB"	FC 144	FC 144
"LS_Calculate_Cylinder"	FC 145	FC 145
"LS2_EOff_MachineOff"	FC 148	FC 148
"LS2_OP_Mode"	FC 149	FC 149
"LS1_Main"	FC 168	FC 168
"LS1_STEPS_BASEPOS"	FC 169	FC 169	// Run on Automatic start UP
"LS1_STEPS_IN"	FC 170	FC 170	// Steps to move a Cylinder in to the storrage
"LS1_STEPS_OUT"	FC 171	FC 171	// Steps to move a cylinder out of the strorrage
"LS2_Main"	FC 188	FC 188
"LS2_STEPS_BASEPOS"	FC 189	FC 189	// Run on Automatic start UP
"LS2_STEPS_IN"	FC 190	FC 190	// Steps to move a Cylinder in to the storrage
"LS2_STEPS_OUT"	FC 191	FC 191	// Steps to move a cylinder out of the strorrage
"LS2_STEPS_PALLETT_CHANGE"	FC 192	FC 192
"LS1_Errors_049-064"	FC 209	FC 209
"LS1_Errors_065-080"	FC 219	FC 219
"Pipe_Magazin_Status"	FC 220	FC 220
"Mark_as_unknown"	FC 221	FC 221
"Mark_as_empty"	FC 222	FC 222
"Mark_as_occupied"	FC 223	FC 223
"LS2_Errors_049-064"	FC 229	FC 229
"LS2_Errors_081-096"	FC 230	FC 230
"LS2_OP_161_176"	FC 235	FC 235
"LS2_Errors_065-080"	FC 239	FC 239
"Fanuc_Control"	FC 300	FC 300
"iPar_ServerMain"	FC 900	FC 900
"iPar_ServerIO12"	FC 901	FC 901
"ROB_RCV_ESTOP"	I 0.0	BOOL
"ROB_RCV_AUTO"	I 0.1	BOOL
"ROB_RCV_AREA_IO1"	I 0.2	BOOL
"ROB_RCV_AREA_IO2"	I 0.3	BOOL
"BarcodeIO1_Ex:Input1"	I 28.0	BOOL	// Level of Ext.In1 of optional connected CMC600
"BarcodeIO1_Ex:Input2"	I 28.1	BOOL	// Level of Ext.In2 of optional connected CMC600
"BarcodeIO1_Sensor1"	I 28.2	BOOL	// Level Sensor 1 of the device
"BarcodeIO1_Sensor2"	I 28.3	BOOL	// Level Sensor 2 of the device
"BarcodeIO1_RD_Toggle"	I 28.7	BOOL	// Is inverted each reading gate
"BarcodeIO1_Ready"	I 29.0	BOOL	// State of the device
"BarcodeIO1_Reserved1"	I 29.1	BOOL
"BarcodeIO1_OK"	I 29.2	BOOL	// Good Read of the last reading result
"BarcodeIO1_NOK"	I 29.3	BOOL	// NoRead of the last reading result
"BarcodeIO1_External_Out1"	I 29.4	BOOL	// State of the device
"BarcodeIO1_External_Out2"	I 29.5	BOOL	// State of the device
"BarcodeIO1_Result1"	I 29.6	BOOL	// Level of Output / Result 1 of the device
"BarcodeIO1_Result2"	I 29.7	BOOL	// Level of Output / Result 2 of the device
"BarcodeIO2_Ex:Input1"	I 38.0	BOOL	// Level of Ext.In1 of optional connected CMC600
"BarcodeIO2_Ex:Input2"	I 38.1	BOOL	// Level of Ext.In2 of optional connected CMC600
"BarcodeIO2_Sensor1"	I 38.2	BOOL	// Level Sensor 1 of the device
"BarcodeIO2_Sensor2"	I 38.3	BOOL	// Level Sensor 2 of the device
"BarcodeIO2_RD_Toggle"	I 38.7	BOOL	// Is inverted each reading gate
"BarcodeIO2_Ready"	I 39.0	BOOL	// State of the device
"BarcodeIO2_Reserved1"	I 39.1	BOOL
"BarcodeIO2_OK"	I 39.2	BOOL	// Good Read of the last reading result
"BarcodeIO2_NOK"	I 39.3	BOOL	// NoRead of the last reading result
"BarcodeIO2_External_Out1"	I 39.4	BOOL	// State of the device
"BarcodeIO2_External_Out2"	I 39.5	BOOL	// State of the device
"BarcodeIO2_Result1"	I 39.6	BOOL	// Level of Output / Result 1 of the device
"BarcodeIO2_Result2"	I 39.7	BOOL	// Level of Output / Result 2 of the device
"IO1_AGV_Request"	I 47.0	BOOL
"IO1_AGV_in_Station"	I 47.1	BOOL
"IO2_AGV_Request"	I 47.4	BOOL
"IO2_AGV_in_Station"	I 47.5	BOOL
"E140_0"	I 140.0	BOOL
"I_CB_24V_OK"	I 140.1	BOOL
"I_CB_Temperature"	I 140.2	BOOL
"I_CB_PhaseOK"	I 140.3	BOOL
"I_CB_Power_LS12"	I 140.4	BOOL
"I_CB_PowerSpare1"	I 140.5	BOOL
"I_CB_PowerSpare2"	I 140.6	BOOL
"E140_7"	I 140.7	BOOL
"CB_BTN_AutoStart"	I 141.0	BOOL
"CB_BTN_Reset"	I 141.1	BOOL
"E141_2"	I 141.2	BOOL
"E141_3"	I 141.3	BOOL
"E141_4"	I 141.4	BOOL
"E141_5"	I 141.5	BOOL
"E141_6"	I 141.6	BOOL
"E141_7"	I 141.7	BOOL
"I_Door1_Closed"	I 142.0	BOOL
"I_Door1_Error"	I 142.1	BOOL
"I_Door1_Btn_White"	I 142.2	BOOL
"I_Door1_Btn_Yellow"	I 142.3	BOOL
"I_Door1_Keyswitch"	I 142.4	BOOL
"I_Door2_Closed"	I 142.5	BOOL
"I_Door2_Error"	I 142.6	BOOL
"I_Door2_Btn_White"	I 142.7	BOOL
"I_Door2_Btn_Yellow"	I 143.0	BOOL
"I_Door2_Keyswitch"	I 143.1	BOOL
"I_Door3_Closed"	I 143.2	BOOL
"I_Door3_Error"	I 143.3	BOOL
"I_Door3_Btn_White"	I 143.4	BOOL
"I_Door3_Btn_Yellow"	I 143.5	BOOL
"I_Door3_Keyswitch"	I 143.6	BOOL
"E143_7"	I 143.7	BOOL
"E144_0"	I 144.0	BOOL
"E144_1"	I 144.1	BOOL
"E144_2"	I 144.2	BOOL
"E144_3"	I 144.3	BOOL
"E144_4"	I 144.4	BOOL
"E144_5"	I 144.5	BOOL
"E144_6"	I 144.6	BOOL
"E144_7"	I 144.7	BOOL
"I_IO1_BTN_Reset"	I 161.1	BOOL
"I_IO2_BTN_Reset"	I 161.3	BOOL
"I_LS01_Gate_Open_NO"	I 164.4	BOOL
"I_LS01_Gate_Open_NC"	I 164.5	BOOL
"I_LS02_Gate_Open_NO"	I 164.6	BOOL
"I_LS02_Gate_Open_NC"	I 164.7	BOOL
"I_LS01_Palet_Controll_34"	I 168.0	BOOL	// LS01 Liniarverstellung: Palettenkontrolle 3+4
"I_LS01_Palet_Controll_12"	I 168.5	BOOL	// LS01 Liniarverstellung: Palettenkontrolle 1+2
"I_LS02_Palet_Controll_12"	I 169.4	BOOL	// LS02 Liniarverstellung: Palettenkontrolle 1+2
"I_LS02_Palet_Control_34"	I 170.3	BOOL	// LS02 Liniarverstellung: Palettenkontrolle 3+4 (laut Schaltplan auf E170.7)
"I_LS02_Palet_Controll_34"	I 170.7	BOOL	// LS02 Liniarverstellung: Palettenkontrolle 3+4
"I_LS01_Shaft_Control_lef"	I 172.0	BOOL	// LS01 Achsenkontrolle links
"I_LS01_Shaft_Control_rig"	I 172.1	BOOL	// LS01 Achsenkontrolle rechts
"I_LS02_Shaft_Control_lef"	I 172.2	BOOL	// LS02 Achsenkontrolle links
"I_LS02_Shaft_Control_rig"	I 172.3	BOOL	// LS02 Achsenkontrolle rechts
"E172_4"	I 172.4	BOOL
"E172_5"	I 172.5	BOOL
"E172_6"	I 172.6	BOOL
"E172_7"	I 172.7	BOOL
"CB_FB_ESTOP_CH1"	I 220.0	BOOL
"CB_FB_ESTOP_CH2"	I 220.1	BOOL
"E220_2"	I 220.2	BOOL
"E220_3"	I 220.3	BOOL
"CB_DOOR1_CH1"	I 225.0	BOOL
"CB_DOOR1_CH2"	I 225.1	BOOL
"CB_DOOR2_CH1"	I 225.2	BOOL
"CB_DOOR2_CH2"	I 225.3	BOOL
"CB_DOOR3_CH1"	I 225.4	BOOL
"CB_DOOR3_CH2"	I 225.5	BOOL
"E225_5"	I 225.6	BOOL
"E225_6"	I 225.7	BOOL
"CB_ESTOP_DDOR_CH1"	I 230.0	BOOL
"CB_ESTOP_DDOR_CH2"	I 230.1	BOOL
"CB_SEL_Automatic"	I 230.2	BOOL
"E230_3"	I 230.3	BOOL
"CB_ESTOP:_Remote_CH1"	I 230.4	BOOL
"CB_ESTOP:_Remote_CH2"	I 230.5	BOOL
"CB_ESTOP_BTN_CH1"	I 230.6	BOOL
"CB_ESTOP_BTN_CH2"	I 230.7	BOOL
"CB_CAR1_Bypass_CH1"	I 235.0	BOOL
"CB_CAR1_Bypass_CH2"	I 235.1	BOOL
"CB_CAR2_Bypass_CH1"	I 235.2	BOOL
"CB_CAR2_Bypass_CH2"	I 235.3	BOOL
"CB_RBG3_Mainainance_CH1"	I 235.4	BOOL
"CB_RBG3_Mainainance_CH2"	I 235.5	BOOL
"CB_RBG1_Bypass_CH1"	I 235.6	BOOL
"CB_RBG1_Bypass_CH2"	I 235.7	BOOL
"CB_RBG2_Bypass_CH1"	I 240.0	BOOL
"CB_RBG2_Bypass_CH2"	I 240.1	BOOL
"CB_RBG3_Bypass_CH1"	I 240.2	BOOL
"CB_RBG3_Bypass_CH2"	I 240.3	BOOL
"CB_RBG1_Mainainance_CH1"	I 240.4	BOOL
"CB_RBG1_Mainainance_CH2"	I 240.5	BOOL
"CB_RBG2_Mainainance_CH1"	I 240.6	BOOL
"CB_RBG2_Mainainance_CH2"	I 240.7	BOOL
"IO1_FB_Power1_CH1"	I 250.0	BOOL
"IO1_FB_Power1_CH2"	I 250.1	BOOL
"IO1_FB_STOP_CH1"	I 250.2	BOOL
"IO1_FB_STOP_CH2"	I 250.3	BOOL
"IO2_FB_Power1_CH1"	I 255.0	BOOL
"IO2_FB_Power1_CH2"	I 255.1	BOOL
"IO2_FB_STOP_CH1"	I 255.2	BOOL
"IO2_FB_STOP_CH2"	I 255.3	BOOL
"CB_DOOR4_OK_CH1"	I 260.0	BOOL
"CB_DOOR4_OK_CH2"	I 260.1	BOOL
"CB_DOOR5_OK_CH1"	I 260.2	BOOL
"CB_DOOR5_OK_CH2"	I 260.3	BOOL
"IO1_LB_OK_CH1"	I 260.4	BOOL
"IO1_LB_OK_CH2"	I 260.5	BOOL
"IO1_LB_Rack_OK_CH1"	I 260.6	BOOL
"IO1_LB_Rack_OK_CH2"	I 260.7	BOOL
"IO2_LB_OK_CH1"	I 265.0	BOOL
"IO2_LB_OK_CH2"	I 265.1	BOOL
"IO2_LB_Rack_OK_CH1"	I 265.2	BOOL
"IO2_LB_Rack_OK_CH2"	I 265.3	BOOL
"IO12_ESTOP_BTN_CH1"	I 265.4	BOOL
"IO12_ESTOP_BTN_CH2"	I 265.5	BOOL
"IO12_ESTOP_DOOR_CH1"	I 265.6	BOOL
"IO12_ESTOP_DOOR_CH2"	I 265.7	BOOL
"IO1_HSCAN_OK_CH1"	I 270.0	BOOL
"IO1_HSCAN_OK_CH2"	I 270.1	BOOL
"IO2_HSCAN_OK_CH1"	I 270.2	BOOL
"IO2_HSCAN_OK_CH2"	I 270.3	BOOL
"E270:4"	I 270.4	BOOL
"E270:5"	I 270.5	BOOL
"IO1_SEL_AUTO"	I 270.6	BOOL
"IO2_SEL_AUTO"	I 270.7	BOOL
"IO1_BYPASS_CH1"	I 275.0	BOOL
"IO1_BYPASS_CH2"	I 275.1	BOOL
"IO2_BYPASS_CH1"	I 275.2	BOOL
"IO2_BYPASS_CH2"	I 275.3	BOOL
"BarcodeIO2_Counter"	IB 391	BYTE
"BarcodeIO2_Length_LOW"	IB 393	BYTE
"BarcodeIO2_Length_HIGH"	IB 394	BYTE
"OFF"	M 0.0	BOOL	// immer aus
"ON"	M 0.1	BOOL	// immer ein
"LS1_ModeService"	M 1.0	BOOL
"LS1_ModeManual"	M 1.1	BOOL
"LS1_ModeAuto"	M 1.2	BOOL
"LS1_ModeBypass"	M 1.3	BOOL
"LS1_LifeBitMasterOK"	M 1.7	BOOL
"LS1_Error"	M 2.2	BOOL
"LS1_DivEoff"	M 2.3	BOOL
"LS1_Eoff"	M 2.4	BOOL
"LS2_LifeBitMasterOK"	M 3.7	BOOL
"LS2_Error"	M 4.2	BOOL
"LS2_DivEoff"	M 4.3	BOOL
"LS2_Eoff"	M 4.4	BOOL
"TR_1_CAR_1"	M 7.0	BOOL
"TR_1_CAR_2"	M 7.1	BOOL
"TR_2_CAR_1"	M 7.2	BOOL
"TR_2_CAR_2"	M 7.3	BOOL
"Clock0_1"	M 10.0	BOOL	// CPU-Takt 0,1s
"Clock0_2"	M 10.1	BOOL	// CPU-Takt 0,2s
"Clock0_4"	M 10.2	BOOL	// CPU-Takt 0,4s
"Clock0_5"	M 10.3	BOOL	// CPU-Takt 0,5s
"Clock0_8"	M 10.4	BOOL	// CPU-Takt 0,8s
"Clock1_0"	M 10.5	BOOL	// CPU-Takt 1,0s
"Clock1_6"	M 10.6	BOOL	// CPU-Takt 1,6s
"Clock2_0"	M 10.7	BOOL	// CPU-Takt 2,0s
"Tick0_1"	M 11.0	BOOL	// Impuls 0,1s
"Tick0_2"	M 11.1	BOOL	// Impuls 0,2s
"Tick0_4"	M 11.2	BOOL	// Impuls 0,4s
"Tick0_5"	M 11.3	BOOL	// Impuls 0,6s
"Tick0_8"	M 11.4	BOOL	// Impuls 0,8s
"Tick1_0"	M 11.5	BOOL	// Impuls 1,0s
"Tick1_6"	M 11.6	BOOL	// Impuls 1,6s
"Tick2_0"	M 11.7	BOOL	// Impuls 2,0s
"SysPulse_0_1"	M 12.0	BOOL
"SysPulse_0_2"	M 12.1	BOOL
"SysPulse_0_4"	M 12.2	BOOL
"SysPulse_0_5"	M 12.3	BOOL
"SysPulse_0_8"	M 12.4	BOOL
"SysPulse_1_0"	M 12.5	BOOL
"SysPulse_1_6"	M 12.6	BOOL
"SysPulse_2_0"	M 12.7	BOOL
"NullBit"	M 20.0	BOOL
"pFl_ModBus1_CLK"	M 32.2	BOOL
"RBG1_ReleaseIO"	M 40.0	BOOL
"RBG2_ReleaseIO"	M 40.1	BOOL
"RBG3_ReleaseIO"	M 40.2	BOOL
"FanucSpare1"	M 400.0	BOOL
"FanucSpare2"	M 400.1	BOOL
"NGAD0"	M 500.0	BOOL
"NGAD1"	M 500.1	BOOL
"TRUE"	M 500.2	BOOL
"FALSE"	M 500.3	BOOL
"IBN-1"	M 501.0	BOOL
"IBN-0"	M 501.1	BOOL
"RC_BTN_3_S1"	M 720.2	BOOL
"RC_BTN_4_S1"	M 720.3	BOOL
"RC_BTN_5_S1"	M 720.4	BOOL
"RC_BTN_6_S1"	M 720.5	BOOL
"RC_BTN_7_S1"	M 720.6	BOOL
"RC_BTN_8_S1"	M 720.7	BOOL
"RC_BTN_9_S1"	M 721.0	BOOL
"RC_BTN_10_S1"	M 721.1	BOOL
"RC_BTN_3_S2"	M 722.2	BOOL
"RC_BTN_4_S2"	M 722.3	BOOL
"RC_BTN_5_S2"	M 722.4	BOOL
"RC_BTN_6_S2"	M 722.5	BOOL
"RC_BTN_7_S2"	M 722.6	BOOL
"RC_BTN_8_S2"	M 722.7	BOOL
"RC_BTN_9_S2"	M 723.0	BOOL
"RC_BTN_10_S2"	M 723.1	BOOL
"RC_pFl_Btn_01"	M 726.0	BOOL
"RC_pFl_Btn_02"	M 726.1	BOOL
"CB_iPar_Check"	M 920.0	BOOL
"CB_iPar_UpLoad_1"	M 920.1	BOOL
"CB_iPar_DownL_1"	M 920.2	BOOL
"CB_iPar_DownL_2"	M 920.3	BOOL
"CB_iPar_ReqDiag"	M 920.5	BOOL
"CB_iPar_UpLoad_2"	M 921.1	BOOL
"pFL_CB_IO_EndWago_1"	M 924.2	BOOL
"pFL_CB_StartWago"	M 925.1	BOOL
"pFL_CB_EndWago_1"	M 925.2	BOOL
"pFL_CB_EndWago_2"	M 925.3	BOOL
"CB_IO_iPar_Check"	M 940.0	BOOL
"CB_IO_iPar_UpLoad_1"	M 940.1	BOOL
"CB_IO_iPar_DownL_1"	M 940.2	BOOL
"CB_IO_iPar_DownL_2"	M 940.3	BOOL
"CB_IO_iPar_ReqDiag"	M 940.5	BOOL
"CB_IO_iPar_UpLoad_2"	M 941.1	BOOL
"pFL_CB_IO_StartWago"	M 945.1	BOOL
"pFL_CB_IO_EndWago_2"	M 945.3	BOOL
"LS1_pFl_12"	M 1201.2	BOOL
"LS1_pFl_13"	M 1201.3	BOOL
"LS1_pFl_14"	M 1201.4	BOOL
"LS1_pFl_15"	M 1201.5	BOOL
"LS1_pFl_16"	M 1201.6	BOOL
"LS2_pFl_12"	M 1202.2	BOOL
"LS2_pFl_13"	M 1202.3	BOOL
"LS2_pFl_14"	M 1202.4	BOOL
"LS2_pFl_15"	M 1202.5	BOOL
"LS2_pFl_16"	M 1202.6	BOOL
"IO1_pFl_Delete_Barcode"	M 1410.0	BOOL
"IO2_pFl_Delete_Barcode"	M 1410.1	BOOL
"IO1_pFl_Save_Barcode"	M 1410.2	BOOL
"IO2_pFl_Save_Barcode"	M 1410.3	BOOL
"Bruno_B"	M 2013.0	BOOL	// Programmpunkt muss noch bearbeitet werden
"bTemp0"	MB 20	BYTE
"diTemp00"	MD 20	DWORD
"CPY_DATETIME_1"	MD 830	DWORD
"CPY_DATETIME_2"	MD 834	DWORD
"iTemp00"	MW 20	WORD
"EMPTY_MAGAZIIN"	MW 50	INT
"LS1_CntMsg"	MW 120	INT
"LS2_CntMsg"	MW 122	INT
"NullWord"	MW 200	WORD
"RC_Select"	MW 724	INT
"CN1_Save_Modb"	MW 1230	INT
"CNT_ModB_1"	MW 1400	INT
"Bruno_W1"	MW 2014	WORD	// Schmierwort
"Bruno_W2"	MW 2016	WORD	// Schmierwort
"Cycle"	OB 1	OB 1
"CYC_INT5"	OB 35	OB 35	// Cyclic Interrupt 5
"I/O_FLT1"	OB 82	OB 82	// I/O Point Fault 1
"I/O_FLT2"	OB 83	OB 83	// I/O Point Fault 2
"OBNL_FLT"	OB 85	OB 85	// OB Not Loaded Fault
"RACK_FLT"	OB 86	OB 86	// Loss of Rack Fault
"COMM_FLT"	OB 87	OB 87	// Communication Fault
"COMPLETE RESTART"	OB 100	OB 100	// Complete Restart
"PROG_ERR"	OB 121	OB 121	// Programming Error
"MOD_ERR"	OB 122	OB 122	// Module Access Error
"ROB_ESTOP"	Q 0.0	BOOL
"ROB_FenceOpen"	Q 0.1	BOOL
"ROB_IO1_OK"	Q 0.2	BOOL
"ROB_I02_OK"	Q 0.3	BOOL
"BarcodeIO1_Trigger"	Q 29.0	BOOL
"BarcodeIO2_Trigger"	Q 39.0	BOOL
"IO1_Permit_AGV"	Q 47.4	BOOL
"IO2_Permit_AGV"	Q 47.5	BOOL
"A140_0"	Q 140.0	BOOL
"O_CB_Reset_24V"	Q 140.1	BOOL
"A140_2"	Q 140.2	BOOL
"A140_3"	Q 140.3	BOOL
"A140_4"	Q 140.4	BOOL
"CB_LP_State_0"	Q 140.5	BOOL
"CB_LP_State_1"	Q 140.6	BOOL
"CB_LP_State_2"	Q 140.7	BOOL
"CB_LP_Start"	Q 141.0	BOOL
"CB_LP_Reset"	Q 141.1	BOOL
"A141_2"	Q 141.2	BOOL
"A141_3"	Q 141.3	BOOL
"A141_4"	Q 141.4	BOOL
"A141_5"	Q 141.5	BOOL
"A141_6"	Q 141.6	BOOL
"A141_7"	Q 141.7	BOOL
"O_Door1_Reset"	Q 142.0	BOOL
"O_Door1_LP_White"	Q 142.1	BOOL
"O_Door1_LP_Yellow"	Q 142.2	BOOL
"O_Door1_Release"	Q 142.3	BOOL
"O_Door2_Reset"	Q 142.4	BOOL
"O_Door2_LP_White"	Q 142.5	BOOL
"O_Door2_LP_Yellow"	Q 142.6	BOOL
"O_Door2_Release"	Q 142.7	BOOL
"O_Door3_Reset"	Q 143.0	BOOL
"O_Door3_LP_White"	Q 143.1	BOOL
"O_Door3_LP_Yellow"	Q 143.2	BOOL
"O_Door3_Release"	Q 143.3	BOOL
"A143.4"	Q 143.4	BOOL
"A143.5"	Q 143.5	BOOL
"A143.6"	Q 143.6	BOOL
"A143.7"	Q 143.7	BOOL
"A144_0"	Q 144.0	BOOL
"A144_1"	Q 144.1	BOOL
"A144_2"	Q 144.2	BOOL
"A144_3"	Q 144.3	BOOL
"A144_4"	Q 144.4	BOOL
"A144_5"	Q 144.5	BOOL
"A144_6"	Q 144.6	BOOL
"A144_7"	Q 144.7	BOOL
"CB_LP_State_0_LS"	Q 165.5	BOOL
"CB_LP_State_1_LS"	Q 165.6	BOOL
"CB_LP_State_2_LS"	Q 165.7	BOOL
"A_132K3_LS1_fast_down"	Q 167.3	BOOL	// Ladestation 1 Hydraulik Lift schnell
"A_142K3_LS2_fast_down"	Q 167.7	BOOL	// Ladestation 2 Hydraulik Lift schnell
"IO1_Power_CH1"	Q 250.0	BOOL
"IO1_Power_CH2"	Q 250.1	BOOL
"IO1_Release_CH1"	Q 250.2	BOOL
"IO1_Release_CH2"	Q 250.3	BOOL
"IO2_Power_CH1"	Q 255.0	BOOL
"IO2_Power_CH2"	Q 255.1	BOOL
"IO2_Release_CH1"	Q 255.2	BOOL
"IO2_Release_CH2"	Q 255.3	BOOL
"TON"	SFB 4	SFB 4	// Generate an On Delay
"USEND"	SFB 8	SFB 8	// Uncoordinated Sending of Data
"URCV"	SFB 9	SFB 9	// Uncoordinated Receiving of Data
"RDREC"	SFB 52	SFB 52	// Read a Process Data Record
"WRREC"	SFB 53	SFB 53	// Write a Process Data Record
"RALRM"	SFB 54	SFB 54	// Receive Alarm Data
"RD_SINFO"	SFC 6	SFC 6	// Read OB Start Information
"DPRD_DAT"	SFC 14	SFC 14	// Read Consistent Data of a Standard DP Slave
"DPWR_DAT"	SFC 15	SFC 15	// Write Consistent Data to a Standard DP Slave
"BLKMOV"	SFC 20	SFC 20	// Copy Variables
"FILL"	SFC 21	SFC 21	// Initialize a Memory Area
"TEST_DB"	SFC 24	SFC 24	// Test Data Block
"DIS_AIRT"	SFC 41	SFC 41	// Delay the Higher Priority Interrupts and Asynchronous Errors
"EN_AIRT"	SFC 42	SFC 42	// Enable Higher Priority Interrupts and Asynchronous Errors
"STP"	SFC 46	SFC 46	// Change the CPU to STOP
"RDSYSST"	SFC 51	SFC 51	// Read a System Status List or Partial List
"WR_USMSG"	SFC 52	SFC 52	// Write a User-Defined Diagnostic Event to the Diagnostic Buffer
"WR_REC"	SFC 58	SFC 58	// Write Data Record
"RD_REC"	SFC 59	SFC 59	// Read a Data Record
"tPlcOn"	T 1	TIMER
"t_Err_012"	T 2	TIMER
"T_CN1_Modb_1"	T 20	TIMER
"T_CN1_Modb_OK"	T 21	TIMER
"t_Err_015"	T 22	TIMER
"LS1_Delay_Start"	T 50	TIMER
"LS2_Delay_Start"	T 51	TIMER
"tDelayDoor"	T 55	TIMER
"LS1_t_DelayReadyOnline"	T 60	TIMER
"LS1_Delay_Error_lift"	T 61	TIMER
"LS1_BasePoswait"	T 89	TIMER
"LS1_Wait_for_Table_out"	T 90	TIMER
"LS1_T_Delay_TableCenter"	T 91	TIMER
"LS1_T_Delay_Measure"	T 92	TIMER
"LS2_T_Delay_Measure"	T 93	TIMER
"LS2_T_Startup_Warning"	T 94	TIMER
"LS1_T_Startup_Horn"	T 95	TIMER
"LS1_SH_occupation_error"	T 96	TIMER
"LS1_Palletsensor_error"	T 97	TIMER
"LS1_Wait_for_Table_in"	T 98	TIMER
"LS1_tAknowl"	T 99	TIMER
"LS2_T_Err_NONC_FS_plus"	T 100	TIMER
"LS2_T_Err_NONC_FS_minus"	T 101	TIMER
"LS2_T_Err_NONC_SH_in_pos"	T 102	TIMER
"t_Timeout_CAR_01"	T 120	TIMER
"t_Timeout_CAR_02"	T 121	TIMER
"t_Timeout_TR_01"	T 122	TIMER
"t_Timeout_TR_02"	T 123	TIMER
"t_Timeout_TR_03"	T 124	TIMER
"t_Timeout_LS_01"	T 125	TIMER
"t_Timeout_LS_02"	T 126	TIMER
"t_Timeout_LS_03"	T 127	TIMER
"t_Timeout_MAIN"	T 128	TIMER
"LS1_T_Err_NONC_FS_plus"	T 150	TIMER
"LS1_T_Err_NONC_FS_minus"	T 151	TIMER
"LS1_T_Err_NONC_SH_in_pos"	T 152	TIMER
"LS2_t_DelayReadyOnline"	T 160	TIMER
"LS2_Delay_Error_lift"	T 161	TIMER
"LS2_BasePoswait"	T 189	TIMER
"LS2_Wait_for_Table_out"	T 190	TIMER
"LS2_T_Delay_TableCenter"	T 191	TIMER
"LS1_T_Startup_Warning"	T 194	TIMER
"LS2_T_Startup_Horn"	T 195	TIMER
"LS2_SH_occupation_error"	T 196	TIMER
"LS2_Palletsensor_error"	T 197	TIMER
"LS2_Wait_for_Table_in"	T 198	TIMER
"LS2_tAknowl"	T 199	TIMER
"Pause_Robot_Pulse"	T 200	TIMER
"OneMove"	UDT 7	UDT 7
"LS_Digital_Inputs"	UDT 80	UDT 80
"LS_Digital_Outputs"	UDT 81	UDT 81
"Digital_InputsSafetydoor"	UDT 82	UDT 82
"Digital_Out_Safetydoor"	UDT 83	UDT 83
"Pipe_Positions"	UDT 200	UDT 200
"Loadingstation_to_PC"	UDT 201	UDT 201
"PC_to_Loadingstation"	UDT 202	UDT 202
"Roboter_Test"	VAT 1	
"Tab_PLC_TO_ROBOT"	VAT 2	
"Tab_ROBOT_TO_PLC"	VAT 3	
"Barcode2"	VAT 4	
"BarcodeTest"	VAT 5	
"Barcode1"	VAT 6	
"LS1 Steps"	VAT 7	
"LS2 Steps"	VAT 8	
"LS2 SICKKamaraIO"	VAT 9	
"VAT_Shaft Control"	VAT 10	
"BarcodeDelete"	VAT 11	
END_SYMBOL_TABLE

SYMBOL_TABLE
"IDB_Safe_Main"	DB 1	FB 1
"DB_TRO"	DB 2	DB 2
"DB_LIF"	DB 3	DB 3
"DB_TEL"	DB 4	DB 4
"DB_BRI"	DB 5	DB 5
"DB_ComGateway"	DB 10	DB 10
"IDB_FB2_TRO"	DB 12	FB 2
"IDB_FB2_LIF"	DB 13	FB 2
"IDB_FB21_TEL"	DB 14	FB 21
"DB_OrderBuffer"	DB 15	DB 15
"DB_IntentData"	DB 17	DB 17
"DB_TargetData"	DB 19	DB 19
"IDB_FB3_TRO"	DB 20	FB 3
"IDB_FB22"	DB 22	FB 22
"IDB_FB29"	DB 29	FB 29
"IDB_MasterInterface"	DB 33	FB 13
"DB_ANALOG"	DB 50	DB 50
"INOUT"	DB 80	DB 80
"DB_ActualHookdata"	DB 92	DB 92	// Hookdata of actual trollayposition
"Moves"	DB 101	DB 101
"DB_STEPS_IBN_Auto_Test"	DB 109	DB 109
"InstanzDB PNIODiag"	DB 126	FB 126
"InstanzDB STATDiag"	DB 127	DB 127
"DB_Crane"	DB 130	DB 130
"DB_Steps"	DB 132	DB 132
"DB_CylinderTypes"	DB 133	DB 133
"DB_Area"	DB 150	DB 150
"IDB_FB190"	DB 190	FB 190
"IDB_FB190_2"	DB 191	FB 190
"IDB1_FB192"	DB 192	FB 192
"IDB1_FB192_2"	DB 193	FB 192
"TRO_Positions"	DB 200	DB 200
"BR01_TR01"	DB 201	DB 201
"BR01_TR02"	DB 202	DB 202
"BR01_TR03"	DB 203	DB 203
"BR01_TR04"	DB 204	DB 204
"BR01_TR05"	DB 205	DB 205
"BR01_TR06"	DB 206	DB 206
"BR01_TR07"	DB 207	DB 207
"BR01_TR08"	DB 208	DB 208
"BR01_TR09"	DB 209	DB 209
"BR01_TR10"	DB 210	DB 210
"BR01_TR11"	DB 211	DB 211
"BR02_TR01"	DB 212	DB 212
"BR02_TR02"	DB 213	DB 213
"BR02_TR03"	DB 214	DB 214
"BR02_TR04"	DB 215	DB 215
"BR02_TR05"	DB 216	DB 216
"BR02_TR06"	DB 217	DB 217
"BR02_TR07"	DB 218	DB 218
"BR02_TR08"	DB 219	DB 219
"BR02_TR09"	DB 220	DB 220
"BR02_TR10"	DB 221	DB 221
"BR02_TR11"	DB 222	DB 222
"BR03_TR01"	DB 223	DB 223
"BR03_TR02"	DB 224	DB 224
"BR03_TR03"	DB 225	DB 225
"BR03_TR04"	DB 226	DB 226
"BR03_TR05"	DB 227	DB 227
"BR03_TR06"	DB 228	DB 228
"BR03_TR07"	DB 229	DB 229
"BR03_TR08"	DB 230	DB 230
"BR03_TR09"	DB 231	DB 231
"BR03_TR10"	DB 232	DB 232
"BR03_TR11"	DB 233	DB 233
"BR04_TR01"	DB 234	DB 234
"BR04_TR02"	DB 235	DB 235
"BR04_TR03"	DB 236	DB 236
"BR04_TR04"	DB 237	DB 237
"BR04_TR05"	DB 238	DB 238
"BR04_TR06"	DB 239	DB 239
"BR04_TR07"	DB 240	DB 240
"BR04_TR08"	DB 241	DB 241
"BR04_TR09"	DB 242	DB 242
"BR04_TR10"	DB 243	DB 243
"BR04_TR11"	DB 244	DB 244
"BR05_TR01"	DB 245	DB 245
"BR05_TR02"	DB 246	DB 246
"BR05_TR03"	DB 247	DB 247
"BR05_TR04"	DB 248	DB 248
"BR05_TR05"	DB 249	DB 249
"BR05_TR06"	DB 250	DB 250
"BR05_TR07"	DB 251	DB 251
"BR05_TR08"	DB 252	DB 252
"BR05_TR09"	DB 253	DB 253
"BR05_TR10"	DB 254	DB 254
"BR05_TR11"	DB 255	DB 255
"BR06_TR01"	DB 256	DB 256
"BR06_TR02"	DB 257	DB 257
"BR06_TR03"	DB 258	DB 258
"BR06_TR04"	DB 259	DB 259
"BR06_TR05"	DB 260	DB 260
"BR06_TR06"	DB 261	DB 261
"BR06_TR07"	DB 262	DB 262
"BR06_TR08"	DB 263	DB 263
"BR06_TR09"	DB 264	DB 264
"BR06_TR10"	DB 265	DB 265
"BR06_TR11"	DB 266	DB 266
"BR07_TR01"	DB 267	DB 267
"BR07_TR02"	DB 268	DB 268
"BR07_TR03"	DB 269	DB 269
"BR07_TR04"	DB 270	DB 270
"BR07_TR05"	DB 271	DB 271
"BR07_TR06"	DB 272	DB 272
"BR07_TR07"	DB 273	DB 273
"BR07_TR08"	DB 274	DB 274
"BR07_TR09"	DB 275	DB 275
"BR07_TR10"	DB 276	DB 276
"BR07_TR11"	DB 277	DB 277
"BR08_TR01"	DB 278	DB 278
"BR08_TR02"	DB 279	DB 279
"BR08_TR03"	DB 280	DB 280
"BR08_TR04"	DB 281	DB 281
"BR08_TR05"	DB 282	DB 282
"BR08_TR06"	DB 283	DB 283
"BR08_TR07"	DB 284	DB 284
"BR08_TR08"	DB 285	DB 285
"BR08_TR09"	DB 286	DB 286
"BR08_TR10"	DB 287	DB 287
"BR08_TR11"	DB 288	DB 288
"BR09_TR01"	DB 289	DB 289
"BR09_TR02"	DB 290	DB 290
"BR09_TR03"	DB 291	DB 291
"BR09_TR04"	DB 292	DB 292
"BR09_TR05"	DB 293	DB 293
"BR09_TR06"	DB 294	DB 294
"BR09_TR07"	DB 295	DB 295
"BR09_TR08"	DB 296	DB 296
"BR09_TR09"	DB 297	DB 297
"BR09_TR10"	DB 298	DB 298
"BR09_TR11"	DB 299	DB 299
"BR10_TR01"	DB 300	DB 300
"BR10_TR02"	DB 301	DB 301
"BR10_TR03"	DB 302	DB 302
"BR10_TR04"	DB 303	DB 303
"BR10_TR05"	DB 304	DB 304
"BR10_TR06"	DB 305	DB 305
"BR10_TR07"	DB 306	DB 306
"BR10_TR08"	DB 307	DB 307
"BR10_TR09"	DB 308	DB 308
"BR10_TR10"	DB 309	DB 309
"BR10_TR11"	DB 310	DB 310
"BR11_TR01"	DB 311	DB 311
"BR11_TR02"	DB 312	DB 312
"LIF_Pos"	DB 350	DB 350
"IDB_Modbus1"	DB 362	FB 102
"ProfiNet"	DB 400	DB 400
"Error_Safety"	DB 410	DB 410
"IDB_ESTOP_1"	DB 450	FB 215
"IDB_ESTOP_2"	DB 451	FB 185
"F_GLOBDB"	DB 545	DB 545	// F_: F_Global_Data Block
"F00035_75x_667_4FDI_4FDO"	DB 555	FB 272
"F00040_75x_667_4FDI_4FDO"	DB 556	FB 272
"F00045_75x_661_4FDI_24V"	DB 557	FB 272
"F00055_75x_667_4FDI_4FDO"	DB 558	FB 272
"F_IO"	DB 690	DB 690
"F_Position"	DB 695	DB 695
"F_GBL_RECV"	DB 750	DB 750
"IDB_F_RCV"	DB 751	FB 226
"F_GBL_SEND"	DB 752	DB 752
"IDB_F_SND"	DB 753	FB 225
"IDB_Axis_Position"	DB 800	FB 5
"IDB_WagoiPar_Rack"	DB 901	FB 37
"IDB_WagoiPar_BRI"	DB 920	FB 37
"IDB_WagoiPar_TRO"	DB 921	FB 37
"IDB_WagoiPar_LIF"	DB 922	FB 37
"DB_iPar_Diag"	DB 930	FB 101
"DIAG_PROFI_V2_iPar"	DB 931	DB 931	// diagnosis data of PROFIsafe modules V2 iPar with FB101
"DB_Vorlage"	DB 999	DB 999
"DB_LS1"	DB 1300	DB 1300
"IDB_LS1_Circum"	DB 1329	FB 29
"DB_LS"	DB 1350	DB 1350
"iPar_Data_Rack"	DB 1901	DB 1901
"iPar_Data_Bridge"	DB 1920	DB 1920
"iPar_Data_Trolley"	DB 1921	DB 1921
"iPar_Data_Lift"	DB 1922	DB 1922
"Safe_Main"	FB 1	FB 1
"MovidriveB_Control"	FB 2	FB 2
"MovidriveC_Control"	FB 3	FB 3
"Axis_Position"	FB 5	FB 5
"MasterInterface"	FB 13	FB 13
"CheckEncoder"	FB 21	FB 21
"GetCircumference"	FB 22	FB 22
"WAGO_Analog_Input_4_20"	FB 29	FB 29	// WAGO A/D-Wandler 4-20mA
"WAGO_iPar_UDL_4_Mod"	FB 37	FB 37	// WAGO up- / download iParameter PROFIsafe Modules
"TSEND"	FB 63	FB 63	// Send Data
"TRCV"	FB 64	FB 64	// Receive Data
"TCON"	FB 65	FB 65	// Connect
"TDISCON"	FB 66	FB 66	// Disconnect
"Safety_Position"	FB 70	FB 70	// Sichere Positionsüberwachung
"Safety_Direction"	FB 72	FB 72	// Sichere Richtungserfassung
"Safety_Speed"	FB 73	FB 73	// Sichere Geschwindigkeit
"Safety_SpeedCheck"	FB 74	FB 74
"Wago_Trolley"	FB 81	FB 81
"F_Input_MAP"	FB 91	FB 91
"ESTOP"	FB 92	FB 92
"GetArea"	FB 95	FB 95
"DiagPROFIsafe_V2_iPar"	FB 101	FB 101	// read diagnosis data of PROFIsafe modules V2 iPar
"MODBUSPN"	FB 102	FB 102	// MODBUS PN CPU
"TCP_COMM"	FB 103	FB 103	// TCP Kommunikation
"MOD_CLI"	FB 104	FB 104
"MOD_SERV"	FB 105	FB 105
"PNIODiag"	FB 126	FB 126	// Profibus/DP und Profinet/IO-Diagnose
"STATDiag"	FB 127	FB 127	// Zweitbaustein (PNIODiag)
"F_TON"	FB 185	FB 185	// F_: Timer Switch On Delay
"F_TOF"	FB 186	FB 186	// F_: Timer Switch Off Delay
"CopyHookDBs"	FB 190	FB 190
"READ_DBL"	FB 192	FB 192	// read db from memorycard
"WRITE_DBL"	FB 193	FB 193	// write db to memorycard
"F_ESTOP1"	FB 215	FB 215	// F_: Emergency Stop / Stop Category 1
"F_ACK_GL"	FB 219	FB 219	// F_: Global Acknowledgement of all F-I/O of a RTG
"F_SENDS7"	FB 225	FB 225	// F_: Send S7 Connection
"F_RCVS7"	FB 226	FB 226	// F_: Receive S7 Connection
"F_IO_CGP"	FB 272	FB 272	// F_: Driver Block In-Output with Channel Granular Passivation
"F_CTRL_1"	FB 273	FB 273
"F_CTRL_2"	FB 274	FB 274	// F_: Test Block an Programm Run Control
"F_DIAG_N"	FB 275	FB 275
"FITON"	FB 276	FB 276
"FITOF"	FB 277	FB 277
"FIACK_GL"	FB 278	FB 278
"F-CALL"	FC 1	FC 1
"Init"	FC 2	FC 2
"AG_SEND"	FC 5	FC 5	// AG SEND
"AG_RECV"	FC 6	FC 6	// AG RECEIVE
"DT_TOD"	FC 8	FC 8	// DT to TOD
"OpHours"	FC 9	FC 9
"EQ_STRNG"	FC 10	FC 10	// Equal String
"AbsEncoder"	FC 11	FC 11
"Motor_2_frequ"	FC 12	FC 12
"DT to DATE"	FC 15	FC 15	// DT to DATE
"Scan_BRI"	FC 21	FC 21
"Scan_BRI_MAN"	FC 22	FC 22	// Scan Bride Manual Mode
"Scan_BRI_DBs"	FC 23	FC 23
"Scan_LIF"	FC 25	FC 25
"Scan_LIF_Man"	FC 26	FC 26
"Scan_TEL"	FC 27	FC 27
"Scan_TEL_Man"	FC 28	FC 28
"SCALE_WAGO_AI"	FC 29	FC 29	// for WAGO 250-466 4-20mA SE Standard
"Inputs"	FC 30	FC 30
"Outputs"	FC 31	FC 31
"MeasureSystem"	FC 33	FC 33
"SEL"	FC 36	FC 36	// Select
"Errors"	FC 40	FC 40
"Errors Reset"	FC 41	FC 41
"Errors_001-016_GEN1"	FC 42	FC 42
"Errors_017-032_GEN2"	FC 43	FC 43
"Errors_033-048_NET"	FC 44	FC 44
"Errors_113-128"	FC 45	FC 45
"Errors_129-144_08"	FC 46	FC 46
"Errors_145-160"	FC 47	FC 47
"EOff_MachineOff"	FC 48	FC 48
"OP_Mode"	FC 49	FC 49
"Send_Buffer"	FC 52	FC 52
"MSG_161-176"	FC 55	FC 55
"MSG_177_192"	FC 56	FC 56
"CableDrum"	FC 60	FC 60
"TargetPosLift"	FC 70	FC 70
"CheckHookType"	FC 72	FC 72
"CheckWindowDi"	FC 100	FC 100
"Communication"	FC 103	FC 103
"STEPS_IBN_AUTO_TEST"	FC 109	FC 109	// Continiues automatictest for comisstioning
"STEPS_Control"	FC 110	FC 110
"STEPS_OrderData"	FC 111	FC 111
"STEPS_BASEPOS"	FC 112	FC 112
"STEPS_EMPTY"	FC 113	FC 113
"STEPS_GET"	FC 114	FC 114
"STEPS_PUT"	FC 115	FC 115
"Axis_TROLLEY"	FC 210	FC 210
"Axis_TROLLEY_Release"	FC 211	FC 211
"Axis_TROLLEY_Control"	FC 212	FC 212
"Axis_TROLLEY_Speed"	FC 213	FC 213
"Axis_TROLLEY_Scan"	FC 214	FC 214
"Axis_TROLLEY_Scan_Man"	FC 215	FC 215
"Axis_TROLLEY_Position"	FC 216	FC 216	// real pos to virtual pos
"Axis_TROLLEY_Flt_065-080"	FC 219	FC 219
"Axis_LIFT"	FC 220	FC 220
"Axis_LIFT_Control"	FC 222	FC 222
"Axis_LIFT_Speed"	FC 223	FC 223
"Axis_LIFT_Scan"	FC 224	FC 224
"Axis_LIFT_Flt_081-096"	FC 229	FC 229
"Axis_TELESCOPES"	FC 230	FC 230
"Axis_TEL_Control"	FC 232	FC 232
"Axis_TEL_Speed"	FC 233	FC 233
"Axis_TEL_Scan"	FC 234	FC 234
"Axis_TEL_Chk"	FC 235	FC 235
"Axis_TEL_Status"	FC 236	FC 236
"Axis_TEL_Mode_Status"	FC 237	FC 237
"Axis_TEL_BCD"	FC 238	FC 238
"Axis_TEL_Flt_097-112"	FC 239	FC 239
"Axis_TEL_Encoder"	FC 240	FC 240
"iPar_ServerCall"	FC 900	FC 900
"Scan_LIF_New"	FC 1025	FC 1025
"Scan_LIF_Man_New"	FC 1026	FC 1026
"TROGetPosVal"	FC 1071	FC 1071
"E   35.0"	I 35.0	BOOL	// spare
"E   35.1"	I 35.1	BOOL	// spare
"I_TRO_FB_Lift"	I 35.2	BOOL	// Feedback safestop lift
"I_TRO_FB_Trolley"	I 35.3	BOOL	// Feedback safestop  trolley
"I_TRO_FB_Telescope"	I 40.0	BOOL	// Feedback safestop no FU
"E   40.1"	I 40.1	BOOL	// spare
"I_TRO_FB_Estop_CH1"	I 40.2	BOOL	// Feedback E-Stop  CH1
"I_TRO_FB_Estop_CH2"	I 40.3	BOOL	// Feedback E-Stop  CH2
"I_TRO_EStop"	I 45.0	BOOL	// Emergency stop activ
"I_TRO_Brake_OK"	I 45.1	BOOL	// Temperature brake resistors OK
"E   45.2"	I 45.2	BOOL	// spare
"E   45.3"	I 45.3	BOOL	// spare
"I_TRO_LIF_Overl_L_NC"	I 55.0	BOOL	// Overload-Monitoring left NC
"I_TRO_LIF_Overl_R_NC"	I 55.1	BOOL	// Overload-Monitoring right NC
"I_TRO_LIF_Slap_L_NC"	I 55.2	BOOL	// Slap-Rope-Monitoring left NC
"I_TRO_LIF_Slap_R_NC"	I 55.3	BOOL	// Slap-Rope-Monitoring right NC
"I_TRO_Fuse_115V_OK"	I 75.0	BOOL	// 115V AC OK
"I_TRO_Fuse_24V_OK"	I 75.1	BOOL	// fuse 24V DC OK
"I_TRO_Overtemp_Cabinet"	I 75.2	BOOL	// high temperature cabinet
"I_TRO_Power Brakes_OK"	I 75.3	BOOL	// Power supply brakes OK
"I_TRO_Power_Lift_OK"	I 75.4	BOOL	// Power supply lift OK
"I_TRO_Power_Drum_OK"	I 75.5	BOOL	// Power supply cable drum OK
"I_TRO_Power_Cabinet_Fan"	I 75.6	BOOL	// Power supply cabinet fan OK
"I_TRO_Cabinet_Fan_On"	I 75.7	BOOL	// 0=cabinet fan running
"I_TRO_BTN_Reset"	I 76.0	BOOL	// Reset button (top cabinet)
"I_TRO_BTN_Preset"	I 76.1	BOOL	// Preset button (3s)
"I_TRO_Preset_Bit_0"	I 76.2	BOOL	// Preset selection switch bit 0
"I_TRO_Preset_Bit_1"	I 76.3	BOOL	// Preset selection switch bit 1
"I_TRO_Preset_Bit_2"	I 76.4	BOOL	// Preset selection switch bit 2
"I_TRO_Preset_Bit_3"	I 76.5	BOOL	// Preset selection switch bit 3
"E 76_6"	I 76.6	BOOL	// spare
"E 76_7"	I 76.7	BOOL	// spare
"I_Check_CableDrum_NO"	I 77.0	BOOL	// check cable drum NO
"I_Check_CableDrum_NC"	I 77.1	BOOL	// check cable drum NC
"E  77_2"	I 77.2	BOOL	// spar
"E  77_3"	I 77.3	BOOL	// spar
"I_Buffer_left_Free"	I 77.4	BOOL	// Buffer left occupied //
"I_Buffer_right_Free"	I 77.5	BOOL	// Buffer right occupied //
"I_LIF_Limit_TOP"	I 77.6	BOOL	// Lift limit switch top (minus)
"I_LIF_Limit_BOTTOM"	I 77.7	BOOL	// Lift limit switch bottom (plus)
"I_LIF_Pos_TOP_NO"	I 78.0	BOOL	// Lift limit prox. top NO
"I_LIF_Pos_TOP_NC"	I 78.1	BOOL	// Lift limit prox. top NC
"I_TRO_Limit_plus"	I 78.2	BOOL	// Tolley limit switch plus
"I_TRO_Limit_minus"	I 78.3	BOOL	// Tolley limit switch minus
"I_TRO_FS_plus_NO"	I 78.4	BOOL	// Tolley prox. switch forced slow plus NO
"I_TRO_FS_plus_NC"	I 78.5	BOOL	// Tolley prox. switch forced slow plus NC
"I_TRO_FS_minus_NO"	I 78.6	BOOL	// Tolley prox. switch forced slow minus NO
"I_TRO_FS_minus_NC"	I 78.7	BOOL	// Tolley prox. switch forced slow minus NC
"I_SSI_Barcode_noPos"	I 79.0	BOOL	// Datamatrix SSI error: no position
"I_SSI_Barcode_dirty"	I 79.1	BOOL	// Datamatrix SSI error: dirty
"I_Profinet_Barcode_noPos"	I 79.2	BOOL	// Datamatrix Profinet error: no position
"I_Profinet_Barcode_dirty"	I 79.3	BOOL	// Datamatrix Profinet error: dirty
"I_TRO_Drop_1_P"	I 79.4	BOOL	// Trolley drop off protection plus 1
"I_TRO_Drop_2_P"	I 79.5	BOOL	// Trolley drop off protection plus 2
"I_TRO_Drop_1_M"	I 79.6	BOOL	// Trolley drop off protection minus 1
"I_TRO_Drop_2_M"	I 79.7	BOOL	// Trolley drop off protection minus 2
"I_TRO_Plus"	I 80.0	BOOL	// Trolley drive plus
"I_TRO_Minus"	I 80.1	BOOL	// Trolley drive minus
"I_Lift_up"	I 80.2	BOOL	// Lift drive up
"I_Lift_down"	I 80.3	BOOL	// Lift drive down
"I_TEL_Plus"	I 80.4	BOOL	// Tellescope drive plus
"I_TEL_Minus"	I 80.5	BOOL	// Telescope drive minus
"E 80_6"	I 80.6	BOOL	// spare
"E 80_7"	I 80.7	BOOL	// spare
"E 85_0"	I 85.0	BOOL	// spare
"E 85_1"	I 85.1	BOOL	// spare
"E 85_2"	I 85.2	BOOL	// spare
"E 85_3"	I 85.3	BOOL	// spare
"I_TEL_Status1"	I 85.4	BOOL	// Drive telescopes status1
"I_TEL_Status2"	I 85.5	BOOL	// Drive telescopes status2
"E 85_6"	I 85.6	BOOL
"E 85_7"	I 85.7	BOOL
"I_LIF_Overload_L_NO"	I 86.0	BOOL	// Overload-Monitoring left NO
"I_LIF_Overload_R_NO"	I 86.1	BOOL	// Overload-Monitoring right NO
"I_LIF_SlapRope_L_NO"	I 86.2	BOOL	// Slap-Rope-Monitoring left NO
"I_LIF_SlapRope_R_NO"	I 86.3	BOOL	// Slap-Rope-Monitoring right NO
"E      86.4"	I 86.4	BOOL	// spare
"E      86.5"	I 86.5	BOOL	// spare
"I_LIF_Front_LastHookOcc"	I 86.6	BOOL	// hook front left occupied long
"I_LIF_Front_FirstHookOcc"	I 86.7	BOOL	// hook rear left occupied short
"I_LIF_Rear_LastHookOcc"	I 87.0	BOOL	// hook front right occupied long
"I_LIF_Rear_FirstHookOcc"	I 87.1	BOOL	// hook rear right occupied short
"E      87.2"	I 87.2	BOOL	// spare
"E      87.3"	I 87.3	BOOL	// spare
"I_TEL_inMidle_L"	I 87.4	BOOL	// telescope left in middle position
"I_TEL_inMidle_R"	I 87.5	BOOL	// telescope right in middle position
"E      87.6"	I 87.6	BOOL
"I_TEL_Left_Occ_NO"	I 87.7	BOOL	// telescope left occupied NO
"E      88.0"	I 88.0	BOOL
"I_TEL_Right_Occ_NO"	I 88.1	BOOL	// telescope right occupied NO
"I_TEL_Limit_front_NO"	I 88.2	BOOL	// telescopes limit switch front NO
"I_TEL_Limit_front_NC"	I 88.3	BOOL	// telescopes limit switch front NC
"I_TEL_Limit_back_NO"	I 88.4	BOOL	// telescopes limit switch back NO
"I_TEL_Limit_back_NC"	I 88.5	BOOL	// telescopes limit switch back NC
"E      88.6"	I 88.6	BOOL	// spare
"E      88.7"	I 88.7	BOOL	// spare
"E      89.0"	I 89.0	BOOL
"E      89.1"	I 89.1	BOOL
"E      89.2"	I 89.2	BOOL
"E      89.3"	I 89.3	BOOL
"E      89.4"	I 89.4	BOOL
"E      89.5"	I 89.5	BOOL
"E      89.6"	I 89.6	BOOL
"E      89.7"	I 89.7	BOOL
"OFF"	M 0.0	BOOL	// immer aus
"ON"	M 0.1	BOOL	// immer ein
"TRUE"	M 0.2	BOOL
"FALSE"	M 0.3	BOOL
"FIRST_RUN"	M 0.7	BOOL
"ModeService"	M 1.0	BOOL
"ModeManual"	M 1.1	BOOL
"ModeAuto"	M 1.2	BOOL
"ModeBypass"	M 1.3	BOOL
"ModeServiceOrManual"	M 1.4	BOOL
"SEW_EmergencyMode"	M 1.5	BOOL
"ModeAutoOrManual"	M 1.6	BOOL
"LifeBitMasterOK"	M 1.7	BOOL
"Eoff"	M 2.0	BOOL
"DivEoff"	M 2.1	BOOL
"Error"	M 2.2	BOOL
"EmOffRelais_delayed"	M 3.0	BOOL
"TRO_pFL_StopOnCarrier"	M 8.0	BOOL
"TRO_StopOnCarrier"	M 8.1	BOOL
"LIF_pFl_manPrevPos"	M 9.0	BOOL
"LIF_pFl_manNextPos"	M 9.1	BOOL
"Tel_pFl_manMinusPos"	M 9.2	BOOL
"Tel_pFl_manPlusPos"	M 9.3	BOOL
"TEL_nFl_CenterPos"	M 9.4	BOOL
"TEL_StopInCenter"	M 9.5	BOOL
"TEL_pFl_StopInCenter"	M 9.6	BOOL
"Clock0_1"	M 10.0	BOOL	// CPU-Takt 0,1s
"Clock0_2"	M 10.1	BOOL	// CPU-Takt 0,2s
"Clock0_4"	M 10.2	BOOL	// CPU-Takt 0,4s
"Clock0_5"	M 10.3	BOOL	// CPU-Takt 0,5s
"Clock0_8"	M 10.4	BOOL	// CPU-Takt 0,8s
"Clock1_0"	M 10.5	BOOL	// CPU-Takt 1,0s
"Clock1_6"	M 10.6	BOOL	// CPU-Takt 1,6s
"Clock2_0"	M 10.7	BOOL	// CPU-Takt 2,0s
"Tick0_1"	M 11.0	BOOL	// Impuls 0,1s
"Tick0_2"	M 11.1	BOOL	// Impuls 0,2s
"Tick0_4"	M 11.2	BOOL	// Impuls 0,4s
"Tick0_5"	M 11.3	BOOL	// Impuls 0,6s
"Tick0_8"	M 11.4	BOOL	// Impuls 0,8s
"Tick1_0"	M 11.5	BOOL	// Impuls 1,0s
"Tick1_6"	M 11.6	BOOL	// Impuls 1,6s
"Tick2_0"	M 11.7	BOOL	// Impuls 2,0s
"SysPulse_0_1"	M 12.0	BOOL
"SysPulse_0_2"	M 12.1	BOOL
"SysPulse_0_4"	M 12.2	BOOL
"SysPulse_0_5"	M 12.3	BOOL
"SysPulse_0_8"	M 12.4	BOOL
"SysPulse_1_0"	M 12.5	BOOL
"SysPulse_1_6"	M 12.6	BOOL
"SysPulse_2_0"	M 12.7	BOOL
"StartModeAuto"	M 13.0	BOOL
"TEL_pFl_Start"	M 19.0	BOOL
"NullBit"	M 20.0	BOOL
"CB_Lamp_Preset"	M 21.0	BOOL
"TEL_Save_Long_POS_front"	M 25.0	BOOL
"TEL_Save_Long_POS_rear"	M 25.1	BOOL
"TrolleyWasOnCarrier"	M 40.0	BOOL
"SendTrolleyWasOnCarrier"	M 40.1	BOOL
"Next_Step"	M 44.0	BOOL
"SingleStep_ON"	M 44.1	BOOL
"One_Single_Step"	M 44.2	BOOL
"TEL_RackPos"	M 55.0	BOOL
"TEL_LS1_Pos"	M 55.1	BOOL
"TEL_LS2_Pos"	M 55.2	BOOL
"TEL_LS3_Pos"	M 55.3	BOOL
"Safety_Tele_Center"	M 152.0	BOOL
"Safety_Tele_Rear"	M 152.1	BOOL
"Safety_Tele_Front"	M 152.2	BOOL
"Safety_Trolley_in_Pos"	M 153.0	BOOL
"Safety_Lift_Top"	M 154.0	BOOL
"Safety_Lift_Over"	M 154.1	BOOL
"Safety_Lift_Under"	M 154.2	BOOL
"Mode_Bypass"	M 200.2	BOOL
"RED_IBN_Test"	M 420.0	BOOL
"bChangeMaster"	M 500.2	BOOL
"bChangeSlave"	M 500.3	BOOL
"bChange"	M 500.4	BOOL
"IBN-0"	M 501.0	BOOL
"IBN-1"	M 501.1	BOOL
"IBN-TEST"	M 501.2	BOOL
"bErrorVirtualE0"	M 504.0	BOOL
"bErrorVirtualE1"	M 504.1	BOOL
"bErrorVirtualE2"	M 504.2	BOOL
"bErrorVirtualE00"	M 504.3	BOOL
"bErrorVirtualE10"	M 504.4	BOOL
"bErrorVirtualE20"	M 504.5	BOOL
"TRO_iPar_Check"	M 921.0	BOOL
"TRO_iPar_UpLoad"	M 921.1	BOOL
"TRO_iPar_DownL"	M 921.2	BOOL
"TRO_iPar_ReqDiag"	M 921.5	BOOL
"LIF_iPar_Check"	M 922.0	BOOL
"LIF_iPar_UpLoad"	M 922.1	BOOL
"LIF_iPar_DownL"	M 922.2	BOOL
"LIF_iPar_ReqDiag"	M 922.5	BOOL
"TRO_pFl_iPar"	M 925.1	BOOL
"LIF_pFl_iPar_1"	M 925.2	BOOL
"LIF_pFl_iPar_2"	M 925.3	BOOL
"PowerFan_pl"	M 1001.0	BOOL
"PowerFan_n"	M 1001.1	BOOL
"P_FL_TeleCheck1"	M 1401.2	BOOL
"N_FL_TeleCheck1"	M 1401.3	BOOL
"P_FL_TeleCheck2"	M 1401.6	BOOL
"N_FL_TeleCheck2"	M 1401.7	BOOL
"TeleCheckErr1"	M 1402.0	BOOL
"TeleCheckErr2"	M 1402.1	BOOL
"TeleCheckErr3"	M 1402.3	BOOL
"TeleCheckErr4"	M 1402.4	BOOL
"Reset_Err"	M 1410.0	BOOL
"Impuls_1"	M 1500.0	BOOL
"Impuls_2"	M 1500.1	BOOL
"Impuls_3"	M 1500.2	BOOL
"Impuls_4"	M 1500.3	BOOL
"Impuls_5"	M 1500.4	BOOL
"Impuls_6"	M 1500.5	BOOL
"Impuls_7"	M 1500.6	BOOL
"Impuls_8"	M 1500.7	BOOL
"DivPos"	MD 510	DWORD
"TEL_SaveTarget"	MW 14	INT
"NullWord"	MW 20	WORD
"PC_MSG_Counter"	MW 120	INT
"ErrorCode"	MW 520	WORD
"CYCL_EXC"	OB 1	OB 1
"CYC_INT5"	OB 35	OB 35	// Cyclic Interrupt 5
"CYCL_FLT"	OB 80	OB 80	// Cycle Time Fault
"I/O_FLT1"	OB 82	OB 82	// I/O Point Fault 1
"I/O_FLT2"	OB 83	OB 83	// I/O Point Fault 2
"OBNL_FLT"	OB 85	OB 85	// OB Not Loaded Fault
"RACK_FLT"	OB 86	OB 86	// Loss of Rack Fault
"COMM_FLT"	OB 87	OB 87	// Communication Fault
"STARTUP"	OB 100	OB 100
"PROG_ERR"	OB 121	OB 121	// Programming Error
"MOD_ERR"	OB 122	OB 122	// Module Access Error
"O_Bypass_RC"	Q 35.0	BOOL	// bypass remote control
"A    35.1"	Q 35.1	BOOL	// spare
"O_SafeStop_Lift"	Q 35.2	BOOL	// safe stop lift
"O_SafeStop_Trolley"	Q 35.3	BOOL	// safe stop trolley
"O_SafeStop_Telecope"	Q 40.0	BOOL	// safe stop telescope
"A    40.1"	Q 40.1	BOOL	// spare
"O_TRO_Stop_CH1"	Q 40.2	BOOL	// E-Stop trolley CH1
"O_TRO_Stop_CH2"	Q 40.3	BOOL	// E-Stop trolley CH2
"O_SafeRelease_Telescope"	Q 55.0	BOOL
"A 75_0"	Q 75.0	BOOL	// spare
"O_TRO_Reset_24V"	Q 75.1	BOOL	// reset 24V fuses
"A 75_2"	Q 75.2	BOOL	// spare
"O_TRO_LP_Reset"	Q 75.3	BOOL	// lamp reset
"A 75_4"	Q 75.4	BOOL	// spare
"O_TRO_CableDrum"	Q 75.5	BOOL	// start cable drum
"O_TRO_EStop_Reset"	Q 75.6	BOOL	// ESTOP reset
"O_TRO_LP_Preset"	Q 75.7	BOOL	// lamp preset
"O_TRO_Horn"	Q 76.0	BOOL	// startup warning
"O_TRO_State_0"	Q 76.1	BOOL	// lamp state 0
"O_TRO_State_1"	Q 76.2	BOOL	// lamp state 1
"O_TRO_state_2"	Q 76.3	BOOL	// lamp state 2
"A      76.4"	Q 76.4	BOOL	// spare
"O_TRO_MoviPLC_Reset"	Q 76.5	BOOL	// reset movi PLC
"O_TRO_EmergencyMode"	Q 76.6	BOOL	// Emergency Mode
"O_LIFT_StartFan"	Q 76.7	BOOL	// start Lift Fan
"O_TRO_EmergencyMode_Fwd"	Q 77.0	BOOL	// Emergency mode forward
"O_TRO_EmergencyMode_Bwd"	Q 77.1	BOOL	// Emergency mode backward
"A      77.2"	Q 77.2	BOOL
"A      77.3"	Q 77.3	BOOL
"A      77.4"	Q 77.4	BOOL
"A      77.5"	Q 77.5	BOOL
"A      77.6"	Q 77.6	BOOL
"A      77.7"	Q 77.7	BOOL
"O_TEL_Mode1"	Q 85.0	BOOL	// telescope mode_1 Service
"O_TEL_Mode2"	Q 85.1	BOOL	// telescope mode_2 Automatic
"O_TEL_Start"	Q 85.2	BOOL	// start telescope
"O_TEL_Reset"	Q 85.3	BOOL	// reset telescope
"O_TEL_BCD_Bit_1"	Q 85.4	BOOL	// telescope BCD Bit_1
"O_TEL_BCD_Bit_2"	Q 85.5	BOOL	// telescope BCD Bit_2
"O_TEL_BCD_Bit_3"	Q 85.6	BOOL	// telescope BCD Bit_3
"O_TEL_BCD_Bit_4"	Q 85.7	BOOL	// telescope BCD Bit_4
"O_TEL_LightFront_Left"	Q 86.0	BOOL	// lightning telescopes front left ON
"O_TEL_LightFront_Right"	Q 86.1	BOOL	// lightning telescopes rear rigth ON
"O_TEL_LightRear_Left"	Q 86.2	BOOL	// lightning telescopes rear left ON
"O_TEL_LightRear_Right"	Q 86.3	BOOL	// lightning telescopes rear rigth ON
"O_TEL_Preset_Encoder"	Q 86.4	BOOL	// Preset Encoder Telescope
"A     86.5"	Q 86.5	BOOL	// spare
"A     86.6"	Q 86.6	BOOL	// spare
"A     86.7"	Q 86.7	BOOL	// spare
"A     87.0"	Q 87.0	BOOL
"A     87.1"	Q 87.1	BOOL
"A     87.2"	Q 87.2	BOOL
"A     87.3"	Q 87.3	BOOL
"A     87.4"	Q 87.4	BOOL
"A     87.5"	Q 87.5	BOOL
"A     87.6"	Q 87.6	BOOL
"A     87.7"	Q 87.7	BOOL
"TON"	SFB 4	SFB 4	// Generate an On Delay
"USEND"	SFB 8	SFB 8	// Uncoordinated Sending of Data
"URCV"	SFB 9	SFB 9	// Uncoordinated Receiving of Data
"RDREC"	SFB 52	SFB 52	// Read a Process Data Record
"WRREC"	SFB 53	SFB 53	// Write a Process Data Record
"RALRM"	SFB 54	SFB 54	// Receive Alarm Data
"RD_SINFO"	SFC 6	SFC 6	// Read OB Start Information
"DPRD_DAT"	SFC 14	SFC 14	// Read Consistent Data of a Standard DP Slave
"DPWR_DAT"	SFC 15	SFC 15	// Write Consistent Data to a Standard DP Slave
"BLKMOV"	SFC 20	SFC 20	// Copy Variables
"FILL"	SFC 21	SFC 21	// Initialize a Memory Area
"TEST_DB"	SFC 24	SFC 24	// Test Data Block
"DIS_AIRT"	SFC 41	SFC 41	// Delay the Higher Priority Interrupts and Asynchronous Errors
"EN_AIRT"	SFC 42	SFC 42	// Enable Higher Priority Interrupts and Asynchronous Errors
"STP"	SFC 46	SFC 46	// Change the CPU to STOP
"RDSYSST"	SFC 51	SFC 51	// Read a System Status List or Partial List
"WR_USMSG"	SFC 52	SFC 52	// Write a User-Defined Diagnostic Event to the Diagnostic Buffer
"WR_REC"	SFC 58	SFC 58	// Write Data Record
"RD_REC"	SFC 59	SFC 59	// Read a Data Record
"RD_DBL"	SFC 83	SFC 83	// Read Data Block from Load Memory
"WRIT_DBL"	SFC 84	SFC 84	// Write Data Block in Load Memory
"tPlcOn"	T 1	TIMER
"tAknowl"	T 2	TIMER
"tTimeout_TRO"	T 26	TIMER
"T_TRO_Preset"	T 30	TIMER
"tTimeout_LIF"	T 36	TIMER
"tTimeout_LIF2"	T 37	TIMER
"T_Startup_Warning"	T 94	TIMER
"T_Delay_Emeg_Mode"	T 110	TIMER
"DEL_No_Order_Running"	T 119	TIMER
"T_Err_TR_Forced_minus"	T 152	TIMER
"T_Err_TR_Forced_plus"	T 153	TIMER
"T_CheckUS"	T 160	TIMER
"T_CheckUS_OK"	T 161	TIMER
"UDT_Any"	UDT 1	UDT 1
"UDT_SysSave"	UDT 2	UDT 2
"OneMove"	UDT 7	UDT 7
"UDT_SEWState"	UDT 11	UDT 11
"UDT_SEWControl"	UDT 12	UDT 12
"TrDataSheet"	UDT 20	UDT 20	// Zuordnung Turm-DBs
"TRODataSheet"	UDT 21	UDT 21
"HookData"	UDT 100	UDT 100
"HookDataSheetNeu"	UDT 101	UDT 101
"HookDataSheet"	UDT 102	UDT 102
"UDT_CylinderType"	UDT 110	UDT 110
"ROW5"	VAT 1	
"IO-Check"	VAT 2	
"ROW4"	VAT 3	
"ROW3"	VAT 4	
"ROW2"	VAT 5	
"ROW1"	VAT 6	
"ROW6"	VAT 7	
"Order"	VAT 8	
"VAT_Sonar"	VAT 9	
"VAT_Bruno"	VAT 10	
"VAT_NewTarget"	VAT 11	
"VAT_TEL_Encoder"	VAT 12	
"VAT_TR_POS_TEST"	VAT 13	
END_SYMBOL_TABLE
